		(* Execute FB *)
		fbCallMethod.nNumberOfInputArguments := nNoOfInputArgs;
		fbCallMethod.pInputArgInfo := ADR(aInputArgInfo);
		fbCallMethod.cbInputArgInfo := (SIZEOF(aInputArgInfo[1])*nNoOfInputArgs);
		fbCallMethod.pInputArgData := ADR(aInputData);
		fbCallMethod.cbInputArgData := nOffset;
		fbCallMethod.nNumberOfOutputArguments := nNoOfOutputArgs; 
		fbCallMethod.pOutputArgInfo := ADR(aOutputArgInfo); 
		fbCallMethod.cbOutputArgInfo := (SIZEOF(aOutputArgInfo[1]) * nNoOfOutputArgs); 
		fbCallMethod.pOutputArgInfoAndData := ADR(stUpdateVehicleReservationDataData.stOutput);
		fbCallMethod.cbOutputArgInfoAndData := SIZEOF(stUpdateVehicleReservationDataData.stOutput);
		
		stUpdateVehicleReservationDataData.iStatus := 1;
		bCallMethod := TRUE;
		
	ELSIF (stUpdateVehicleReservationDataData.iStatus = 1) THEN
		// Method call Completed...
		IF (eStateMethod = E_TrackClientState.Connected) THEN
			// Method call OK
			IF (stUpdateVehicleReservationDataData.stOutput.eStatus = E_MMServerStatus.eMMServerStatus_Success) THEN
				// Method returned OK
				stUpdateVehicleReservationDataData.iStatus := 2;
				// Trig vehicle data reading because data has changed
				M_VehicleToReadAdd(nVehicleID);
				
			ELSE
				// Method returned with error
				stUpdateVehicleReservationDataData.iStatus := 3;
				stUpdateVehicleReservationDataData.stOutput.sMessage;

			END_IF

		ELSIF (eStateMethod = E_TrackClientState.Error) THEN
			// Method call failed
			stUpdateVehicleReservationDataData.iStatus := 3;

		END_IF
		
	END_IF
ELSE
	M_CallUpdateVehicleReservationData := -1;
	RETURN;

END_IF

M_CallUpdateVehicleReservationData := stUpdateVehicleReservationDataData.iStatus;
END_METHOD

METHOD M_CallUpdateVehicleReworkData : INT
VAR_INPUT
	nVehicleID			: UINT;										(* Magnemotion Vehicle ID *)
	sCarrierID			: STRING(30);								(* Carrier ID *)
	bNOK				: BOOL;										(* TRUE signals that rework is required *)
END_VAR
VAR
END_VAR
IF (stUpdateVehicleReworkDataData.iStatus = 2) OR (stUpdateVehicleReworkDataData.iStatus = 3) THEN
	stUpdateVehicleReworkDataData.iStatus := 0;
END_IF

IF (bConnectedMethod AND NOT bBusyMethod) THEN
	IF (stUpdateVehicleReworkDataData.iStatus = 0) THEN
	(* Setup method calling parameters *)
		(* Method identifier *)
		sObjectIDentifier := stUpdateVehicleReworkDataData.sObjectID;
		sMethodIdentifier := stUpdateVehicleReworkDataData.sMethodID;
	
		(* Method Inputs *)
		stUpdateVehicleReworkDataData.stInput.sCarrierID := sCarrierID;
		stUpdateVehicleReworkDataData.stInput.bNOK := bNOK;
		
		(* Fill input data area with method arguments *)
		MEMSET(ADR(aInputData), 0 ,SIZEOF(aInputData));
		nOffset := 0;
		nOffset := nOffset + MEMCPY(ADR(aInputData)+nOffset, ADR(stUpdateVehicleReworkDataData.stInput),	MIN(SIZEOF(stUpdateVehicleReworkDataData.stInput), (SIZEOF(aInputData)-nOffset)) );
		(* Number of input arguments *)
		nNoOfInputArgs := stUpdateVehicleReworkDataData.iNoOfInputArgs;
		(* Set up input argument information *)
		MEMSET(ADR(aInputArgInfo), 0, SIZEOF(aInputArgInfo));
		aInputArgInfo[1].DataType := eUAType_String;
		aInputArgInfo[1].ValueRank := -1;	// -1: Scalar 
		aInputArgInfo[1].nLenData := SIZEOF(stUpdateVehicleReworkDataData.stInput.sCarrierID);
		aInputArgInfo[2].DataType := eUAType_Boolean;
		aInputArgInfo[2].ValueRank := -1;	// -1: Scalar 
		aInputArgInfo[2].nLenData := SIZEOF(stUpdateVehicleReworkDataData.stInput.bNOK);
		
		(* Method outputs *)
		(* Clear output data area *)
		(* Number of output arguments *)
		nNoOfOutputArgs := stUpdateVehicleReworkDataData.iNoOfOutputArgs;
		(* Set up output argument information *)
		MEMSET(ADR(aOutputArgInfo), 0, SIZEOF(aOutputArgInfo));
		aOutputArgInfo[1].DataType := eUAType_Uint16;
		aOutputArgInfo[1].ValueRank := -1;
		aOutputArgInfo[1].nLenData := SIZEOF(stUpdateVehicleReworkDataData.stOutput.eStatus);
		aOutputArgInfo[2].DataType := eUAType_String;
		aOutputArgInfo[2].ValueRank := -1;
		aOutputArgInfo[2].nLenData := SIZEOF(stUpdateVehicleReworkDataData.stOutput.sMessage);
		(* Set up output  *)
		MEMSET(ADR(stUpdateVehicleReworkDataData.stOutput), 0, SIZEOF(stUpdateVehicleReworkDataData.stOutput));
		stUpdateVehicleReworkDataData.stOutput.nNumberOfOutputArguments := nNoOfOutputArgs;
		stUpdateVehicleReworkDataData.stOutput.stOutputArgInfo[1] := aOutputArgInfo[1];
		stUpdateVehicleReworkDataData.stOutput.stOutputArgInfo[2] := aOutputArgInfo[2];
	
		(* Execute FB *)
		fbCallMethod.nNumberOfInputArguments := nNoOfInputArgs;
		fbCallMethod.pInputArgInfo := ADR(aInputArgInfo);
		fbCallMethod.cbInputArgInfo := (SIZEOF(aInputArgInfo[1])*nNoOfInputArgs);
		fbCallMethod.pInputArgData := ADR(aInputData);
		fbCallMethod.cbInputArgData := nOffset;
		fbCallMethod.nNumberOfOutputArguments := nNoOfOutputArgs; 
		fbCallMethod.pOutputArgInfo := ADR(aOutputArgInfo); 
		fbCallMethod.cbOutputArgInfo := (SIZEOF(aOutputArgInfo[1]) * nNoOfOutputArgs); 
		fbCallMethod.pOutputArgInfoAndData := ADR(stUpdateVehicleReworkDataData.stOutput);
		fbCallMethod.cbOutputArgInfoAndData := SIZEOF(stUpdateVehicleReworkDataData.stOutput);
		
		stUpdateVehicleReworkDataData.iStatus := 1;
		bCallMethod := TRUE;
		
	ELSIF (stUpdateVehicleReworkDataData.iStatus = 1) THEN
		// Method call Completed...
		IF (eStateMethod = E_TrackClientState.Connected) THEN
			// Method call OK
			IF (stUpdateVehicleReworkDataData.stOutput.eStatus = E_MMServerStatus.eMMServerStatus_Success) THEN
				// Method returned OK
				stUpdateVehicleReworkDataData.iStatus := 2;
				// Trig vehicle data reading because data has changed
				M_VehicleToReadAdd(nVehicleID);
								
			ELSE
				// Method returned with error
				stUpdateVehicleReworkDataData.iStatus := 3;
				stUpdateVehicleReworkDataData.stOutput.sMessage;
				
			END_IF
			
		ELSIF (eStateMethod = E_TrackClientState.Error) THEN
			// Method call failed
			stUpdateVehicleReworkDataData.iStatus := 3;

		END_IF
		
	END_IF
ELSE
	M_CallUpdateVehicleReworkData := -1;
	RETURN;

END_IF

M_CallUpdateVehicleReworkData := stUpdateVehicleReworkDataData.iStatus;
END_METHOD

METHOD PROTECTED M_CarrierIDToVehicleID : UINT
VAR_INPUT
	sCarrierID		: STRING(30);
END_VAR

VAR
	i: INT;
END_VAR

// Find vehicle with specified Carrier ID
FOR i := 1 TO MM_MAX_NUMBER_OF_VEHICLE_ELEMENTS BY 1 DO
	IF (aReadVehicleData[i].stVehicle.bDataValid) THEN
		IF (F_StringCompNoCase(aReadVehicleData[i].stVehicle.sCarrierID, sCarrierID) ) THEN
			M_CarrierIDToVehicleID := aReadVehicleData[i].stVehicle.nVehicleID;
			RETURN;
		END_IF
	END_IF
END_FOR

// Not found!
M_CarrierIDToVehicleID := 0;
END_METHOD

/// Check if a specified station index belongs to this cell
METHOD PROTECTED M_CheckStationIndex : BOOL
VAR_INPUT
	iStationNo		: UINT;
END_VAR
VAR
	i				: UINT;
END_VAR

FOR i := 1 TO 5 BY 1 DO
	IF (aStations[i].bPresent) THEN
		IF (iThisStationIndex[i] = iStationNo) THEN
			// Station index found
			M_CheckStationIndex := TRUE;
			RETURN;			
		END_IF
	END_IF
END_FOR

// Not found
M_CheckStationIndex := FALSE;
RETURN;
END_METHOD

/// Check if indexes are found for all specified stations
METHOD PROTECTED M_CheckStationsRead : BOOL
VAR
	i				: UINT;
	bReturn			: BOOL;
END_VAR

bReturn := TRUE;

FOR i := 1 TO 5 BY 1 DO
	IF (aStations[i].bPresent) THEN
		IF (iThisStationIndex[i] > 0) THEN
			// Station index found
		ELSE
			// Index for this station is not found!
			bReturn := FALSE;
			EXIT;
		END_IF
	END_IF
END_FOR

// Not found
M_CheckStationsRead := bReturn;
RETURN;
END_METHOD

/// Check if specified vehicle is Owned by this cell and is to be read (evet-driven reading)
METHOD PROTECTED M_CheckVehicleEventRead : BOOL
VAR_INPUT
	iVehicleNo		: UINT;		// MagneMotion Vehicle number
END_VAR
VAR
	i				: UINT;
	bVehicleOwned	: BOOL;
	bVehicleDoRead	: BOOL;
END_VAR

FOR i := 1 TO MM_MAX_NUMBER_OF_VEHICLE_ELEMENTS BY 1 DO
	IF (anVehiclesToRead[i] = iVehicleNo) THEN
		// Vehicle is found in to-read list
		M_CheckVehicleEventRead := TRUE;
		RETURN;
	END_IF

END_FOR

// Not found
M_CheckVehicleEventRead := FALSE;
RETURN;
END_METHOD

/// Check if specified vehicle is Owned by this cell
METHOD PROTECTED M_CheckVehicleOwned : BOOL
VAR_INPUT
	iVehicleNo		: UINT;		// MagneMotion Vehicle number
END_VAR
VAR
	i				: UINT;
END_VAR

FOR i := 1 TO MM_MAX_NUMBER_OF_VEHICLE_ELEMENTS BY 1 DO
	IF (aReadCellData.stCell.anVehicles[i] = iVehicleNo) THEN
		// Vehicle is found
		M_CheckVehicleOwned := TRUE;
		RETURN;
	END_IF
END_FOR

// Not found
M_CheckVehicleOwned := FALSE;
RETURN;
END_METHOD

/// Check if specified vehicle is survailed by this cell
METHOD PROTECTED M_CheckVehicleSurvail : BOOL
VAR_INPUT
	iVehicleNo		: UINT;		// MagneMotion Vehicle number
END_VAR
VAR
	i				: UINT;
END_VAR

FOR i := 1 TO MM_MAX_NUMBER_OF_VEHICLE_ELEMENTS BY 1 DO
	IF (anExtraVehicles[i] = iVehicleNo) THEN
		// Vehicle is found
		M_CheckVehicleSurvail := TRUE;
		RETURN;
	END_IF
END_FOR

// Not found
M_CheckVehicleSurvail := FALSE;
RETURN;
END_METHOD

METHOD M_ClearAll : BOOL
VAR_INPUT
END_VAR
VAR
	i	: UINT;
END_VAR

//Clear data on station(s)
FOR i:=1 TO 5 DO
	IF aStations[i].bPresent THEN
		// Station data
		aStations[i].stStationData1.nTicket := 0;
		aStations[i].stStationData1.nTicketSize := 0;
		aStations[i].stStationData1.CurrentPriority := 0;
		aStations[i].stStationData1.nCurrentVehicleID := 0;
		aStations[i].stStationData1.nReservedVehicleID := 0;
		aStations[i].stStationData2.nTicket := 0;
		aStations[i].stStationData2.nTicketSize := 0;
		aStations[i].stStationData2.CurrentPriority := 0;
		aStations[i].stStationData2.nCurrentVehicleID := 0;
		aStations[i].stStationData2.nReservedVehicleID := 0;
		
		// Station in/output
		bReadyStationIn[i] := FALSE;
		bReadyStationOut[i] := FALSE;

	END_IF
END_FOR

M_ClearAll := TRUE;
END_METHOD

METHOD PROTECTED M_CommandData
VAR_INPUT
END_VAR
VAR
	i			: USINT;
	iRes		: UINT;
END_VAR
// Handle the command data from OPC UA (stCommand)

CASE eCommandDataState OF
	// Init state
	E_CommandDataState.Undefined:
		eCommandDataState := E_CommandDataState.CheckRequest;		

	// Check command data request
	E_CommandDataState.CheckRequest:
		IF ((stCommand.ChangeRequest <> stStatus.ChangeStatus) AND (stCommand.ChangeRequest > 0)) THEN
			// Check if changes is allowed on mapping data (from LC)
			IF (stAdditionalDataIn.MESHandShakes.DataChangeStatusTransportStatus = stStatus.DataChange) THEN
// NOTE: Changed to match new LC software!!! - Hack!				
//				stStatus.ChangeAcknowledge := stCommand.ChangeRequest;
//				stStatus.DataChange := stStatus.DataChange + 1;
			
				// Find vehicle ID for specified Carrier ID
				iCommandDataVehicleID := M_CarrierIDToVehicleID(stCommand.CarrierID);
				IF ((iCommandDataVehicleID > 0) AND (iCommandDataVehicleID <= MM_MAX_NUMBER_OF_VEHICLE_ELEMENTS)) THEN
					// Specified vehicle found
					IF (F_StringCompNoCase(aReadVehicleData[iCommandDataVehicleID].stVehicle.sOwnerCell, sCellID)) THEN
						// Vehicle belongs to this cell
						stStatus.ValidRequest := TRUE;
						IF (stCommand.Ticket <= 0) THEN
							// Clear reservation data for this carrier (do not add reservation)
							eCommandDataState := E_CommandDataState.UpdateJobData;
						ELSE
							// Add reservation to track server
							eCommandDataState := E_CommandDataState.AddReservation;
						END_IF
					ELSE
						eCommandDataState := E_CommandDataState.Error;
					END_IF
				ELSE
					eCommandDataState := E_CommandDataState.Error;
				END_IF
			END_IF
		END_IF
		
	E_CommandDataState.AddReservation:
		iRes := M_CallAddReservation(	sStationID := stCommand.TargetStation,
										sCarrierID := stCommand.CarrierID,
										nTicket := stCommand.Ticket,
										nTicketSize := stCommand.CarriersInPackage,
										nPriority := stCommand.Priority 	);
		IF (iRes = 2) THEN
			// Success
			eCommandDataState := E_CommandDataState.UpdateJobData;
		ELSIF (iRes = 3) THEN
			// Error!
			F_LogLine('ERROR: AddReservation (Ticket: %d)', stCommand.Ticket);
			eCommandDataState := E_CommandDataState.Error;
		END_IF
	
	E_CommandDataState.UpdateJobData:
		iRes := M_CallUpdateVehicleReservationData(	nVehicleID := iCommandDataVehicleID,
													sTargetStationID := stCommand.TargetStation,
													sCarrierID := stCommand.CarrierID,
													nTicket := stCommand.Ticket,
													nCarriersInPackage := stCommand.CarriersInPackage,
													nPriority := stCommand.Priority,
													sJobID := stCommand.JobID 	);
		IF (iRes = 2) THEN
			// Success
			eCommandDataState := E_CommandDataState.Done;
		ELSIF (iRes = 3) THEN
			// Error!
			F_LogLine('ERROR: UpdateJobData (Ticket: %d)', stCommand.Ticket);
			eCommandDataState := E_CommandDataState.Error;
		END_IF
	
	E_CommandDataState.Done:
		stStatus.LatestTicket := stCommand.Ticket;
		stStatus.NumberOfCarriers := stCommand.CarriersInPackage;
		stStatus.ChangeStatus := stCommand.ChangeRequest;
// NOTE: Changed to match new LC software!!! - Hack!				
		stStatus.ChangeAcknowledge := stCommand.ChangeRequest;
		stStatus.DataChange := stStatus.DataChange + 1;
		eCommandDataState := E_CommandDataState.Undefined;
		
	E_CommandDataState.Error:
		stStatus.ValidRequest := FALSE;
		stStatus.ChangeStatus := stCommand.ChangeRequest;
// NOTE: Changed to match new LC software!!! - Hack!				
		stStatus.ChangeAcknowledge := stCommand.ChangeRequest;
		stStatus.DataChange := stStatus.DataChange + 1;
		eCommandDataState := E_CommandDataState.Undefined;
		
END_CASE
END_METHOD

/// Copy vehicle and ticket information from Source to Target and DELETES information on Source!!
METHOD PROTECTED M_CopyAndClearBufferData : BOOL
VAR_IN_OUT
	stSource		: ST_MMBuffer;
	stTarget		: ST_MMBuffer;
END_VAR

	// Update data for target location
	stTarget.nTicket := stSource.nTicket;
	stTarget.nTicketSize := stSource.nTicketSize;
	stTarget.CurrentPriority := stSource.CurrentPriority;
	stTarget.nReservedVehicleID := stSource.nReservedVehicleID;
	stTarget.nCurrentVehicleID := stSource.nCurrentVehicleID;
	// Clear data for source location
	stSource.nTicket := 0;
	stSource.nTicketSize := 0;
	stSource.CurrentPriority := 0;
	stSource.nCurrentVehicleID := 0;
	stSource.nReservedVehicleID := 0;
END_METHOD

/// Copy vehicle and ticket information from Source to Target and DELETES information on Source!!
METHOD PROTECTED M_CopyBufferData : BOOL
VAR_IN_OUT
	stSource		: ST_MMBuffer;
	stTarget		: ST_MMBuffer;
END_VAR

	// Update data for target location
	stTarget.nTicket := stSource.nTicket;
	stTarget.nTicketSize := stSource.nTicketSize;
	stTarget.CurrentPriority := stSource.CurrentPriority;
	stTarget.nReservedVehicleID := stSource.nReservedVehicleID;
	stTarget.nCurrentVehicleID := stSource.nCurrentVehicleID;
END_METHOD

// Set path to control from this cell
METHOD PUBLIC M_DefinePath : BOOL
VAR_INPUT
	nPathNo				: UINT;		// Path number
END_VAR
VAR
	i					: UINT;
	bFound				: BOOL;
END_VAR

bFound := FALSE;

IF ( (nPathNo > 0) AND (nPathNo <= MM_MAX_NUMBER_OF_PATH_ELEMENTS) ) THEN
	FOR i := 1 TO MM_MAX_NUMBER_OF_PATH_ELEMENTS BY 1 DO
		IF (aPaths[i] = nPathNo) THEN
			// Same path found
			IF (bFound) THEN
				// Already added to list, but found again, delete old value
				aPaths[i] := 0;
			END_IF
			bFound := TRUE;
		ELSIF ( (aPaths[i] = 0) AND NOT bFound ) THEN
			// Free spot found, assign value
			aPaths[i] := nPathNo;
			bFound := TRUE;
		END_IF
	END_FOR
END_IF

M_DefinePath := bFound;
END_METHOD

METHOD PUBLIC M_DefinePathSegment : BOOL
VAR_INPUT
	nPathSegmentNo	: UINT;
	nPathID			: UINT;		// Path number
	rPositionBegin	: REAL;		// Distance on the specified path to begin segment
	rPositionEnd	: REAL;		// Distance on the specified path to end segment
END_VAR
// Check if data is valid
IF ( (nPathID > 0) AND (rPositionBegin >= 0.0) AND (rPositionEnd > rPositionBegin) ) THEN
	IF (nPathSegmentNo = 1) THEN
		stExitPointSeg1LocBegin.nPathID := nPathID;
		stExitPointSeg1LocBegin.fPosition := rPositionBegin;
		stExitPointSeg1LocEnd.nPathID := nPathID;
		stExitPointSeg1LocEnd.fPosition := rPositionEnd;
		M_DefinePathSegment := TRUE;
		
	ELSIF (nPathSegmentNo = 2) THEN
		stExitPointSeg2LocBegin.nPathID := nPathID;
		stExitPointSeg2LocBegin.fPosition := rPositionBegin;
		stExitPointSeg2LocEnd.nPathID := nPathID;
		stExitPointSeg2LocEnd.fPosition := rPositionEnd;
		M_DefinePathSegment := TRUE;
		
	ELSE
		M_DefinePathSegment := FALSE;
		
	END_IF

ELSE
	M_DefinePathSegment := FALSE;
	
END_IF
END_METHOD

// Set data for traffic light
METHOD PUBLIC M_DefineStation : BOOL
VAR_INPUT
	nStationNo			: UINT(1..5);
	sStationID			: STRING(30);
	nLoc1PathID			: UINT;		// Path number for input location
	rLoc1Position		: REAL;		// Distance on the specified path for input location
	nLoc2PathID			: UINT;		// Path number for output location (0 if single station)
	rLoc2Position		: REAL;		// Distance on the specified path for output location (0.0 if single station)
	nLocDecPathID		: UINT;		// Path number for decision point location
	rLocDecPosition		: REAL;		// Distance on the specified path for decision point location
	nPreBufferSize		: UINT;		// Size of pre buffer (number of positions)
	nPostBufferSize		: UINT;		// Size of post buffer (number of positions)
END_VAR
VAR
	i					: UINT;
	bReInit				: BOOL;
END_VAR
IF ( (nLoc1PathID > 0) AND (rLoc1Position >= 0.0) AND
//	 (nLoc2PathID > 0) AND (rLoc2Position >= 0.0) AND	// Allow single position stations!
	 (nLocDecPathID > 0) AND (rLocDecPosition >= 0.0) AND 
	 (nStationNo >= 1) AND (nStationNo <= 5) AND
	 (sStationID <> '') ) THEN
	
	IF ( (aStations[nStationNo].sStationID <> sStationID) OR
		 (aStations[nStationNo].stStationData1.stLocation.nPathID <> nLoc1PathID) OR
		 (aStations[nStationNo].stStationData1.stLocation.fPosition <> rLoc1Position) OR
		 (aStations[nStationNo].stStationData2.stLocation.nPathID <> nLoc2PathID) OR
		 (aStations[nStationNo].stStationData2.stLocation.fPosition <> rLoc2Position) OR
		 (aStations[nStationNo].stDecisionLocation.nPathID <> nLocDecPathID) OR
		 (aStations[nStationNo].stDecisionLocation.fPosition <> rLocDecPosition) OR
		 (aStations[nStationNo].bPresent = FALSE) ) THEN
		
		bReInit := TRUE;
	END_IF

	aStations[nStationNo].sStationID := sStationID;
	aStations[nStationNo].stStationData1.stLocation.nPathID := nLoc1PathID;
	aStations[nStationNo].stStationData1.stLocation.fPosition := rLoc1Position;
	IF (nLoc1PathID > 0) THEN
		aStations[nStationNo].stStationData1.bPresent := TRUE;
	ELSE
		aStations[nStationNo].stStationData1.bPresent := FALSE;		
	END_IF
	aStations[nStationNo].stStationData2.stLocation.nPathID := nLoc2PathID;
	aStations[nStationNo].stStationData2.stLocation.fPosition := rLoc2Position;
	IF (nLoc2PathID > 0) THEN
		aStations[nStationNo].stStationData2.bPresent := TRUE;
	ELSE
		aStations[nStationNo].stStationData2.bPresent := FALSE;		
	END_IF
	aStations[nStationNo].stDecisionLocation.nPathID := nLocDecPathID;
	aStations[nStationNo].stDecisionLocation.fPosition := rLocDecPosition;

	// Buffers	
	FOR i := 1 TO MM_MAX_BUFFER_INDEX BY 1 DO
		IF ( (aStations[nStationNo].astPreBuffer[i].bPresent <> (i <= nPreBufferSize)) OR
			 (aStations[nStationNo].astPostBuffer[i].bPresent <> (i <= nPostBufferSize)) ) THEN
			bReInit := TRUE;
		END_IF
		aStations[nStationNo].astPreBuffer[i].bPresent := (i <= nPreBufferSize);
		aStations[nStationNo].astPostBuffer[i].bPresent := (i <= nPostBufferSize);
	END_FOR
	aStations[nStationNo].bPresent := TRUE;
	
	M_DefineStation := TRUE;
ELSE
	M_DefineStation := FALSE;
END_IF
END_METHOD

// Set data for traffic light
METHOD PUBLIC M_DefineStationBufferAdjust : BOOL
VAR_INPUT
	nStationNo			: UINT(1..5);
	rPreBufferAdjust	: REAL;		// Distance to adjust pre-buffer position (M) - Should be negative for pre-buffer
	rPostBufferAdjust	: REAL;		// Distance to adjust post-buffer position (M) - Should be negative for pre-buffer
END_VAR
VAR
END_VAR
IF ( (nStationNo > 0) AND (nStationNo <= 5) ) THEN
	IF (aStations[nStationNo].bPresent) THEN
		// Station defined
		aStationPreBufAdj[nStationNo] := rPreBufferAdjust;
		aStationPostBufAdj[nStationNo] := rPostBufferAdjust;
		M_DefineStationBufferAdjust := TRUE;
	ELSE
		// Station not defined
		M_DefineStationBufferAdjust := FALSE;
	END_IF
ELSE
	// Outside range
	M_DefineStationBufferAdjust := FALSE;
END_IF
END_METHOD

// Set data for traffic light
METHOD PUBLIC M_DefineTrafficLight : BOOL
VAR_INPUT
	nTrafficLightNo	: UINT;
	nPathID			: UINT;		// Path number
	rPosition		: REAL;		// Distance on the specified path
END_VAR

IF ((nTrafficLightNo > 0) AND (nPathID > 0) AND (rPosition >= 0.0)) THEN
	IF (nTrafficLightNo = 1) THEN
		stTrafficLightLocation.nPathID := nPathID;
		stTrafficLightLocation.fPosition := rPosition;
		M_DefineTrafficLight := TRUE;

	ELSIF (nTrafficLightNo = 2) THEN
		stTrafficLight2Location.nPathID := nPathID;
		stTrafficLight2Location.fPosition := rPosition;
		M_DefineTrafficLight := TRUE;

	ELSE
		M_DefineTrafficLight := FALSE;
		
	END_IF
ELSE
	M_DefineTrafficLight := FALSE;
	
END_IF
END_METHOD

// Set data for enable/disable station
METHOD PUBLIC M_EnableStation : BOOL
VAR_INPUT
	nStationNo			: UINT(1..5);
	bPresent			: BOOL;
END_VAR
VAR
	i					: UINT;
END_VAR
IF (nStationNo <= 5) THEN
	aStations[nStationNo].bPresent := bPresent;
	
	M_EnableStation := TRUE;
ELSE
	M_EnableStation := FALSE;
END_IF
END_METHOD

METHOD PROTECTED M_ErrorWarning
VAR_INPUT
END_VAR
VAR
	bDataChange:BOOL;
END_VAR

bDataChange S= 
M_ErrorWarningObj(arErrorWaringData:= stErrorWarning.ErrorWarningData,
	bActive:= eTrackState = E_TrackState.Error, 
	iErrorWarningType:= 2, 
	diErrorWarningID:= E_AlarmCategory.TrackClient + 0, 
	sDeviceID:= 'Track Client',
	iSeverity:= 2, 
	iNativeID:= 0, 
	sNativeMessage:= 'Error State Machine');
	
bDataChange S= 
M_ErrorWarningObj(arErrorWaringData:= stErrorWarning.ErrorWarningData,
	bActive:= eStateMethod = E_TrackState.Error, 
	iErrorWarningType:= 2, 
	diErrorWarningID:= E_AlarmCategory.TrackClient + 1, 
	sDeviceID:= 'Track Client',
	iSeverity:= 2, 
	iNativeID:= 0, 
	sNativeMessage:= 'Error State Machine Method');
	
bDataChange S= 
M_ErrorWarningObj(arErrorWaringData:= stErrorWarning.ErrorWarningData,
	bActive:= eStateNode = E_TrackState.Error, 
	iErrorWarningType:= 2, 
	diErrorWarningID:= E_AlarmCategory.TrackClient + 2, 
	sDeviceID:= 'Track Client',
	iSeverity:= 2, 
	iNativeID:= 0, 
	sNativeMessage:= 'Error State Machine Node ADS');


stErrorWarning.DataChange := stErrorWarning.DataChange + TO_UINT(bDataChange);
bDataChange := FALSE;
END_METHOD

METHOD M_ErrorWarningObj : BOOL
VAR_INPUT
	bActive				: BOOL;
	iErrorWarningType	: UINT;
	diErrorWarningID 	: UDINT;
	sDeviceID			: STRING(30);
	iSeverity			: UINT;
	iNativeID			: UDINT;
	sNativeMessage		: STRING(80);
END_VAR
VAR_IN_OUT
	arErrorWaringData	: ARRAY [1..255] OF ST_ErrorWarningDataX;
END_VAR
VAR
	iFoundPos			: UINT;
	i					: UINT;
	j					: UINT;
END_VAR
//Look through array to find existing record(s)
FOR i := 1 TO 255 DO
	IF arErrorWaringData[i].ErrorWarningID = 0 THEN
		EXIT;
	END_IF
	//Existing alarm - first
	IF arErrorWaringData[i].ErrorWarningID = diErrorWarningID AND iFoundPos = 0 THEN
		iFoundPos := i;
	//Multiple records - delete
	ELSIF arErrorWaringData[i].ErrorWarningID = diErrorWarningID AND iFoundPos <> 0 THEN
		MEMSET(ADR(arErrorWaringData[i]), 0, SIZEOF(arErrorWaringData[i]));
		M_ErrorWarningObj := TRUE;
	END_IF
END_FOR

//Alarm high
IF bActive THEN
	//New alarm
	IF iFoundPos = 0 THEN
		arErrorWaringData[i].ErrorWarningType := iErrorWarningType;
		arErrorWaringData[i].DeviceID := sDeviceID;
		arErrorWaringData[i].Severity := iSeverity;
		arErrorWaringData[i].NativeID := iNativeID;
		arErrorWaringData[i].NativeMessage := sNativeMessage;
		arErrorWaringData[i].ErrorWarningID := diErrorWarningID;
		arErrorWaringData[i].DateTime := SYSTEMTIME_TO_STRING(fbGetTime.TIMESTR);
		M_ErrorWarningObj := TRUE;
	END_IF
	
//Alarm low
ELSIF NOT bActive AND iFoundPos <> 0 THEN
	MEMSET(ADR(arErrorWaringData[iFoundPos]), 0, SIZEOF(arErrorWaringData[iFoundPos]));
	M_ErrorWarningObj := TRUE;
END_IF

//Defrag
IF M_ErrorWarningObj THEN
	FOR i:= 1 TO 254 DO
		//Find first empty spot
		IF arErrorWaringData[i].ErrorWarningID = 0 THEN
			//Find first record
			FOR j:= i TO 255 DO
				IF arErrorWaringData[j].ErrorWarningID <> 0 THEN
					//Move to empty spot
					arErrorWaringData[i] := arErrorWaringData[j];
					MEMSET(ADR(arErrorWaringData[j]), 0, SIZEOF(arErrorWaringData[j]));
					EXIT;
				END_IF
			END_FOR
		END_IF
		//No more records
		IF j >= 255 THEN
			RETURN;
		END_IF
	END_FOR
END_IF
END_METHOD

/// Add vehicle to be survailed
METHOD PROTECTED M_ExtraVehicleAdd : BOOL
VAR_INPUT
	iVehicleNo		: UINT;
END_VAR
VAR
	i				: UINT;
	bAdded			: BOOL;
	bRemoved		: BOOL;
END_VAR

FOR i := 1 TO MM_MAX_NUMBER_OF_VEHICLE_ELEMENTS BY 1 DO
	// Check if already excists in list
	IF (anExtraVehicles[i] = iVehicleNo) THEN
		anExtraVehicles[i] := 0;
		bRemoved := TRUE;
	END_IF
	// Add to list
	IF ( (NOT bAdded) AND (anExtraVehicles[i] = 0) ) THEN
		anExtraVehicles[i] := iVehicleNo;
		bAdded := TRUE;
	END_IF
	// Check if finished
	IF (bAdded AND bRemoved) THEN
		M_ExtraVehicleAdd := TRUE;
		RETURN;
	END_IF
	
END_FOR

IF (bAdded) THEN
	// Added
	M_ExtraVehicleAdd := TRUE;
	RETURN;
ELSE
	// NOT Added (list is maybe full!)
	M_ExtraVehicleAdd := FALSE;
	RETURN;	
END_IF
END_METHOD

/// Remove vehicle from surveillance list
METHOD PROTECTED M_ExtraVehicleRemove : BOOL
VAR_INPUT
	iVehicleNo		: UINT;
END_VAR
VAR
	i				: UINT;
END_VAR

FOR i := 1 TO MM_MAX_NUMBER_OF_VEHICLE_ELEMENTS BY 1 DO
	IF (anExtraVehicles[i] = iVehicleNo) THEN
		anExtraVehicles[i] := 0;
		M_ExtraVehicleRemove := TRUE;
		RETURN;
	END_IF
END_FOR

// Not found
M_ExtraVehicleRemove := FALSE;
RETURN;
END_METHOD

METHOD PROTECTED M_Init : BOOL
VAR_INPUT
END_VAR
VAR
	i : UINT;
	sTemp : STRING;
END_VAR
IF (NOT bInitDone) THEN
// Client information to stations
	FOR i := 1 TO 5 BY 1 DO
		aStations[i].sCellID := sCellID;
	END_FOR

// OPC UA Method calling information
	(* Use no encryption *)
	stConnectInfoMethod.eSecurityMode 			:= eUASecurityMsgMode_None;
	(*  *)
	stConnectInfoMethod.eSecurityPolicyUri		:= eUASecurityPolicy_None;
	(* USe TCP transport profile *)
	stConnectInfoMethod.eTransportProfileUri	:= eUATransportProfileUri_UATcp;
	(* Application name *)
	stConnectInfoMethod.sApplicationName		:= '';
	(* Connection timeout *)
	stConnectInfoMethod.tConnectTimeout			:= T#1M;
	(* Session timeout *)
	stConnectInfoMethod.tSessionTimeout			:= T#10M;
	(* Method node ID *)
	stObjectNodeID.eIdentifierType				:= E_UAIdentifierType.eUAIdentifierType_String;
	stMethodNodeID.eIdentifierType				:= E_UAIdentifierType.eUAIdentifierType_String;
	(* Method data *)
	M_InitMethodData();
	
// OPC UA Node reading information
	(* Use no encryption *)
	stConnectInfoNodes.eSecurityMode 			:= eUASecurityMsgMode_None;
	(*  *)
	stConnectInfoNodes.eSecurityPolicyUri		:= eUASecurityPolicy_None;
	(* USe TCP transport profile *)
	stConnectInfoNodes.eTransportProfileUri		:= eUATransportProfileUri_UATcp;
	(* Application name *)
	stConnectInfoNodes.sApplicationName			:= '';
	(* Connection timeout *)
	stConnectInfoNodes.tConnectTimeout			:= T#1M;
	(* Session timeout *)
	stConnectInfoNodes.tSessionTimeout			:= T#10M;

	
	bInitDone := TRUE;
END_IF
END_METHOD

METHOD PROTECTED M_InitMethodData : BOOL

(* Method data *)
stAddStationDoubleData.iStatus				:= 0;
stAddStationSingleData.iStatus				:= 0;
stEnableStationData.iStatus					:= 0;
stRemoveStationData.iStatus					:= 0;

stGetCellIndexData.iStatus					:= 0;

stAddPathData.iStatus						:= 0;
stRemovePathData.iStatus					:= 0;
stStartPathData.iStatus						:= 0;
stResetPathData.iStatus						:= 0;
stSuspendPathData.iStatus					:= 0;
stResumePathData.iStatus					:= 0;

stAddTrafficLightData.iStatus				:= 0;
stRemoveTrafficLightData.iStatus			:= 0;
stTrafficLightColorData.iStatus				:= 0;
stSetTrafficLightColorData.iStatus			:= 0;

stMoveToStationInData.iStatus				:= 0;
stMoveToStationOutData.iStatus				:= 0;
stMoveToPositionData.iStatus				:= 0;
stMoveToBufferData.iStatus					:= 0;
stMoveToDecisionPointData.iStatus			:= 0;
stMoveToScannerData.iStatus					:= 0;

//stUpdateVehicleDataData.iStatus			:= 0;
stUpdateVehicleReservationDataData.iStatus	:= 0;
stUpdateVehicleMappingDataData.iStatus		:= 0;
stUpdateVehicleReworkDataData.iStatus		:= 0;
END_METHOD

METHOD PROTECTED M_InitNodeData : BOOL
VAR
	i				: UINT;
	sPrefix 		: STRING;
	
	bReturn			: BOOL;
END_VAR

(* Node data, init to use string identifier and set namespace index *)
FOR i:=1 TO nMaxNodeIDsInList BY 1 DO
	aNodeIDs[i].eIdentifierType := eUAIdentifierType_String;
	aNodeIDs[i].nNamespaceIndex := nNameSpaceIndexNodes;
END_FOR

nNoOfNodes := 0;
cbDataTotal := 0;

// TEST
//eReadType := E_OPC_NodeType.Nodes;
//iReadIndex := 1;

// Comm type selection
CASE eReadType OF
	E_OPC_NodeType.Vehicles:
		// Select vehicle to read data from
		REPEAT
			iReadIndex := iReadIndex+1;
			IF (iReadIndex > MM_MAX_NUMBER_OF_VEHICLE_ELEMENTS) THEN
				EXIT;
			END_IF
			UNTIL (aReadCellData.stCell.anVehicles[iReadIndex] > 0)
		END_REPEAT
		IF (iReadIndex <= MM_MAX_NUMBER_OF_VEHICLE_ELEMENTS) THEN
			// Build remote symbol name
			sPrefix := CONCAT(sObjectIDentifier, '.stTrackStatus');
			// Data pointer for received data
			pReadNodeData := ADR(aReadVehicleData[iReadIndex]);
			// Header data size
			cbDataTotal := SIZEOF(aReadVehicleData[iReadIndex].stReadListReturnInfo);
			
			// Specify nodes to read by variable name
			nNoOfNodes := nNoOfNodes + 1;
			aNodeIDs[nNoOfNodes].sIdentifier := CONCAT(sPrefix, '.aVehicles[');
			aNodeIDs[nNoOfNodes].sIdentifier := CONCAT(aNodeIDs[nNoOfNodes].sIdentifier, UINT_TO_STRING(aReadCellData.stCell.anVehicles[iReadIndex]));
			aNodeIDs[nNoOfNodes].sIdentifier := CONCAT(aNodeIDs[nNoOfNodes].sIdentifier, ']');
			acbDatas[nNoOfNodes] := SIZEOF(aReadVehicleData[iReadIndex]);
			cbDataTotal := cbDataTotal + acbDatas[nNoOfNodes];
			bReturn := TRUE;
		ELSE
			// Read next type
			iReadIndex := 0;
			eReadType := E_OPC_NodeType.Paths;
			bReturn := FALSE;
		END_IF			
		
	E_OPC_NodeType.Paths:
		// Select path to read data from
		REPEAT
			iReadIndex := iReadIndex+1;
			IF (iReadIndex > MM_MAX_NUMBER_OF_PATH_ELEMENTS) THEN
				EXIT;
			END_IF
			UNTIL (abControlledPaths[i])
		END_REPEAT
		IF (iReadIndex <= MM_MAX_NUMBER_OF_PATH_ELEMENTS) THEN
			// Build remote symbol name
			sPrefix := CONCAT(sObjectIDentifier, '.stTrackStatus');
			// Data pointer for received data
			pReadNodeData := ADR(aReadPathData[iReadIndex]);
			// Header data size
			cbDataTotal := SIZEOF(aReadPathData[iReadIndex].stReadListReturnInfo);
			
			// Specify nodes to read by variable name
			nNoOfNodes := nNoOfNodes + 1;
			aNodeIDs[nNoOfNodes].sIdentifier := CONCAT(sPrefix, '.aPaths[');
			aNodeIDs[nNoOfNodes].sIdentifier := CONCAT(aNodeIDs[nNoOfNodes].sIdentifier, UINT_TO_STRING(iReadIndex));
			aNodeIDs[nNoOfNodes].sIdentifier := CONCAT(aNodeIDs[nNoOfNodes].sIdentifier, ']');
			acbDatas[nNoOfNodes] := SIZEOF(aReadPathData[iReadIndex]);
			cbDataTotal := cbDataTotal + acbDatas[nNoOfNodes];
			bReturn := TRUE;
		ELSE
			// Read next type
			iReadIndex := 0;
			eReadType := E_OPC_NodeType.Stations;
			bReturn := FALSE;
		END_IF
		
	E_OPC_NodeType.Stations:
		// Select Station to read data from
		iReadIndex := iReadIndex+1;
		IF (iReadIndex <= MM_MAX_NUMBER_OF_STATION_ELEMENTS) THEN
			// Build remote symbol name
			sPrefix := CONCAT(sObjectIDentifier, '.stTrackStatus');
			// Data pointer
			pReadNodeData := ADR(aReadStationData[iReadIndex]);
			
			// Header data
			cbDataTotal := SIZEOF(aReadStationData[iReadIndex].stReadListReturnInfo);
			
			// Specify nodes to read by variable name
			nNoOfNodes := nNoOfNodes + 1;
			aNodeIDs[nNoOfNodes].sIdentifier := CONCAT(sPrefix, '.aStations[');
			aNodeIDs[nNoOfNodes].sIdentifier := CONCAT(aNodeIDs[nNoOfNodes].sIdentifier, UINT_TO_STRING(iReadIndex));
			aNodeIDs[nNoOfNodes].sIdentifier := CONCAT(aNodeIDs[nNoOfNodes].sIdentifier, ']');
			acbDatas[nNoOfNodes] := SIZEOF(aReadStationData[iReadIndex].stStationData);
			cbDataTotal := cbDataTotal + acbDatas[nNoOfNodes];
			bReturn := TRUE;
		ELSE
			// Read next type
			iReadIndex := 0;
			eReadType := E_OPC_NodeType.Cells;
			bReturn := FALSE;
		END_IF
		
	E_OPC_NodeType.Cells:
		// Select cell status to read data from
		iReadIndex := iThisCellIndex;
		IF (iReadIndex > 0 AND iReadIndex <= MM_MAX_NUMBER_OF_STATION_ELEMENTS) THEN
			// Build remote symbol name
			sPrefix := CONCAT(sObjectIDentifier, '.stTrackStatus');
			// Data pointer
			pReadNodeData := ADR(aReadCellData);
			
			// Header data
			cbDataTotal := SIZEOF(aReadCellData.stReadListReturnInfo);
			
			// Specify nodes to read by variable name
			nNoOfNodes := nNoOfNodes + 1;
			aNodeIDs[nNoOfNodes].sIdentifier := CONCAT(sPrefix, '.aCells[');
			aNodeIDs[nNoOfNodes].sIdentifier := CONCAT(aNodeIDs[nNoOfNodes].sIdentifier, UINT_TO_STRING(iReadIndex));
			aNodeIDs[nNoOfNodes].sIdentifier := CONCAT(aNodeIDs[nNoOfNodes].sIdentifier, ']');
			acbDatas[nNoOfNodes] := SIZEOF(aReadCellData.stCell);
			cbDataTotal := cbDataTotal + acbDatas[nNoOfNodes]; 
			bReturn := TRUE;

			// continue to next type after this read!
			iReadIndex := 0;
			eReadType := E_OPC_NodeType.Vehicles;
		ELSE
			// Read next type
			iReadIndex := 0;
			eReadType := E_OPC_NodeType.Vehicles;
			bReturn := FALSE;
		END_IF
	
END_CASE
END_METHOD

METHOD PROTECTED M_InitNodeData_ADS : BOOL
VAR
	i				: UINT;
	sPrefix 		: STRING;
	
	bReturn			: BOOL;
END_VAR

nNoOfNodes := 0;
cbDataTotal := 0;

// TEST NEW
IF ( (nDecisionPointVehicleNo > 0) AND bReadDecPointVehicle ) THEN
	// Read data from vehicle at decision point (Higher priority!)
	// Build remote symbol name
	sPrefix := CONCAT(sObjectIDentifier, '.stTrackStatus');
	// Data pointer for received data
	pReadNodeData := ADR(aReadVehicleData[nDecisionPointVehicleNo].stVehicle);
	// Header data size
	cbDataTotal := SIZEOF(aReadVehicleData[nDecisionPointVehicleNo].stVehicle);
	
	// Specify nodes to read by variable name
	sTrackServerSymbol := CONCAT(sPrefix, '.aVehicles[');
	sTrackServerSymbol := CONCAT(sTrackServerSymbol, UINT_TO_STRING(nDecisionPointVehicleNo));
	sTrackServerSymbol := CONCAT(sTrackServerSymbol, ']');

	// Remove this vehicle from the event-driven reading list (to make sure it is not continously read!)
	M_VehicleToReadRemove(nDecisionPointVehicleNo);
				
	bReadDecPointVehicle := FALSE;	// Done in M_StateMachineNode_ADS
	bReadDecPointVehicleBusy := TRUE;
	bReturn := TRUE;

	M_InitNodeData_ADS := bReturn;
	RETURN;
END_IF
// END TEST NEW

// Comm type selection
CASE eReadType OF
	E_OPC_NodeType.Vehicles:
		IF ( (nDecisionPointVehicleNo > 0) AND bReadDecPointVehicle ) THEN
			// Read data from vehicle at decision point (Higher priority!)
			// Build remote symbol name
			sPrefix := CONCAT(sObjectIDentifier, '.stTrackStatus');
			// Data pointer for received data
			pReadNodeData := ADR(aReadVehicleData[nDecisionPointVehicleNo].stVehicle);
			// Header data size
			cbDataTotal := SIZEOF(aReadVehicleData[nDecisionPointVehicleNo].stVehicle);
			
			// Specify nodes to read by variable name
			sTrackServerSymbol := CONCAT(sPrefix, '.aVehicles[');
			sTrackServerSymbol := CONCAT(sTrackServerSymbol, UINT_TO_STRING(nDecisionPointVehicleNo));
			sTrackServerSymbol := CONCAT(sTrackServerSymbol, ']');

			// Remove this vehicle from the event-driven reading list (to make sure it is not continously read!)
			M_VehicleToReadRemove(nDecisionPointVehicleNo);
				
			bReadDecPointVehicle := FALSE;	// Done in M_StateMachineNode_ADS
			bReadDecPointVehicleBusy := TRUE;
			bReturn := TRUE;			
		ELSE
	// NEW!!!
			// NOTE: iReadIndex is MagneMotion vehicle No
			REPEAT
				iReadIndex := iReadIndex + 1;
				IF (M_CheckVehicleOwned(iReadIndex)) THEN
					// Vehicle is owned by this cell... Read data from Track Server for this vehicle
					IF (M_CheckVehicleEventRead(iReadIndex)) THEN
						// Vehicle data is selected to be read! (event-based reading)
						EXIT;
					END_IF
				ELSIF (M_CheckVehicleSurvail(iReadIndex)) THEN
					// Vehicle is survailed by this cell (read data continously!)... Read data from Track Server for this vehicle
					EXIT;
				ELSIF (iReadIndex <> nDecisionPointVehicleNo) THEN
					// Not owned or surveilled or being handled by decision point. Delete any previous read data
					IF (iReadIndex > 0 AND iReadIndex <= MM_MAX_NUMBER_OF_VEHICLE_ELEMENTS) THEN
						aReadVehicleData[iReadIndex].stVehicle.bDataValid := FALSE;
					END_IF
				END_IF
				UNTIL (iReadIndex >= MM_MAX_NUMBER_OF_VEHICLE_ELEMENTS)
			END_REPEAT
			
			IF (iReadIndex <= MM_MAX_NUMBER_OF_VEHICLE_ELEMENTS) THEN
				// Build remote symbol name
				sPrefix := CONCAT(sObjectIDentifier, '.stTrackStatus');
				// Data pointer for received data
				pReadNodeData := ADR(aReadVehicleData[iReadIndex].stVehicle);
				// Header data size
				cbDataTotal := SIZEOF(aReadVehicleData[iReadIndex].stVehicle);
				
				// Specify nodes to read by variable name
				sTrackServerSymbol := CONCAT(sPrefix, '.aVehicles[');
				sTrackServerSymbol := CONCAT(sTrackServerSymbol, UINT_TO_STRING(iReadIndex));
				sTrackServerSymbol := CONCAT(sTrackServerSymbol, ']');
				
				// Remove this vehicle from the event-driven reading list
				M_VehicleToReadRemove(iReadIndex);
				
				bReturn := TRUE;
			ELSE
				// Read next type
				iReadIndex := 0;
				eReadType := E_OPC_NodeType.Paths;
				bReturn := FALSE;
			END_IF
	// NEW END!!!	
			// Select vehicle to read data from (only the vehicles this cell is responsible for)
(*			REPEAT
				iReadIndex := iReadIndex+1;
				IF (iReadIndex > MM_MAX_NUMBER_OF_VEHICLE_ELEMENTS) THEN
					EXIT;
				END_IF
				UNTIL (aReadCellData.stCell.anVehicles[iReadIndex] > 0)
			END_REPEAT
			IF (iReadIndex <= MM_MAX_NUMBER_OF_VEHICLE_ELEMENTS) THEN
				// Build remote symbol name
				sPrefix := CONCAT(sObjectIDentifier, '.stTrackStatus');
				// Data pointer for received data
				pReadNodeData := ADR(aReadVehicleData[aReadCellData.stCell.anVehicles[iReadIndex]].stVehicle);
				// Header data size
				cbDataTotal := SIZEOF(aReadVehicleData[aReadCellData.stCell.anVehicles[iReadIndex]].stVehicle);
				
				// Specify nodes to read by variable name
				sTrackServerSymbol := CONCAT(sPrefix, '.aVehicles[');
				sTrackServerSymbol := CONCAT(sTrackServerSymbol, UINT_TO_STRING(aReadCellData.stCell.anVehicles[iReadIndex]));
				sTrackServerSymbol := CONCAT(sTrackServerSymbol, ']');
				bReturn := TRUE;
			ELSE
				// Read next type
				iReadIndex := 0;
				eReadType := E_OPC_NodeType.Paths;
				bReturn := FALSE;
			END_IF		*)
		END_IF
		
	E_OPC_NodeType.Paths:
		// Select path to read data from
		REPEAT
			iReadIndex := iReadIndex+1;
			IF (iReadIndex > MM_MAX_NUMBER_OF_PATH_ELEMENTS) THEN
				EXIT;
			END_IF
			UNTIL (abControlledPaths[iReadIndex])
		END_REPEAT
		IF ((iReadIndex <= MM_MAX_NUMBER_OF_PATH_ELEMENTS) AND NOT tonSkipPathRead.Q) THEN	// Skip path reading when paths are started!
			// Build remote symbol name
			sPrefix := CONCAT(sObjectIDentifier, '.stTrackStatus');
			// Data pointer for received data
			pReadNodeData := ADR(aReadPathData[iReadIndex].stPathData);
			// Header data size
			cbDataTotal := SIZEOF(aReadPathData[iReadIndex].stPathData);
			
			// Specify nodes to read by variable name
			sTrackServerSymbol := CONCAT(sPrefix, '.aPaths[');
			sTrackServerSymbol := CONCAT(sTrackServerSymbol, UINT_TO_STRING(iReadIndex));
			sTrackServerSymbol := CONCAT(sTrackServerSymbol, ']');
			bReturn := TRUE;
		ELSE
			// Read next type
			iReadIndex := 0;
			eReadType := E_OPC_NodeType.Stations;
			bReturn := FALSE;
		END_IF
		
	E_OPC_NodeType.Stations:
		// Select Station to read data from
// TEST
		IF (M_CheckStationsRead()) THEN
			// Index for station data from track server has been found... Only read these stations
			REPEAT
				iReadIndex := iReadIndex+1;
				IF (iReadIndex > MM_MAX_NUMBER_OF_STATION_ELEMENTS) THEN
					EXIT;
				END_IF
				UNTIL (M_CheckStationIndex(iReadIndex))
			END_REPEAT
		ELSE
			// Index for station data from track server has NOT been found... Read data from all stations
			iReadIndex := iReadIndex + 1;
		END_IF
// TEST END
//		iReadIndex := iReadIndex+1;
		IF (iReadIndex <= MM_MAX_NUMBER_OF_STATION_ELEMENTS) THEN
			// Build remote symbol name
			sPrefix := CONCAT(sObjectIDentifier, '.stTrackStatus');
			// Data pointer
			pReadNodeData := ADR(aReadStationData[iReadIndex].stStationData);
			// Header data
			cbDataTotal := SIZEOF(aReadStationData[iReadIndex].stStationData);
			
			// Specify nodes to read by variable name
			sTrackServerSymbol := CONCAT(sPrefix, '.aStations[');
			sTrackServerSymbol := CONCAT(sTrackServerSymbol, UINT_TO_STRING(iReadIndex));
			sTrackServerSymbol := CONCAT(sTrackServerSymbol, ']');
			bReturn := TRUE;
		ELSE
			// Read next type
			iReadIndex := 0;
			eReadType := E_OPC_NodeType.Cells;
			bReturn := FALSE;
		END_IF
	
	E_OPC_NodeType.Cells:
		// Select Station to read data from
		iReadIndex := iThisCellIndex;
		IF (iReadIndex > 0 AND iReadIndex <= MM_MAX_NUMBER_OF_CELL_ELEMENTS) THEN
			// Build remote symbol name
			sPrefix := CONCAT(sObjectIDentifier, '.stTrackStatus');
			// Data pointer
			pReadNodeData := ADR(aReadCellData.stCell);
			// Header data
			cbDataTotal := SIZEOF(aReadCellData.stCell);
			
			// Specify nodes to read by variable name
			sTrackServerSymbol := CONCAT(sPrefix, '.aCells[');
			sTrackServerSymbol := CONCAT(sTrackServerSymbol, UINT_TO_STRING(iReadIndex));
			sTrackServerSymbol := CONCAT(sTrackServerSymbol, ']');
			bReturn := TRUE;

			// continue to next type after this read!
			iReadIndex := 0;
			bReadDecPointVehicle := TRUE;	// Force reading of the vehicle at decision point before other vehicles
			IF (NOT bReadDecPointCellDone) THEN
				bReadDecPointCell := TRUE;
			END_IF
			eReadType := E_OPC_NodeType.Vehicles;
		ELSE
			// Read next type
			iReadIndex := 0;
			bReadDecPointVehicle := TRUE;	// Force reading of the vehicle at decision point before other vehicles
			eReadType := E_OPC_NodeType.Vehicles;
			bReturn := FALSE;
		END_IF

END_CASE

M_InitNodeData_ADS := bReturn;
END_METHOD

METHOD PROTECTED M_InitNodeData_OPCUA : BOOL
VAR
	i		: UINT;
	sPrefix : STRING;
END_VAR
VAR
	cbDataTotal2 : UINT;
END_VAR
// NOTE!!!
// Maximum of 10 elements to read for each Node List reading!


(* Node data, init to use string identifier and set namespace index *)
FOR i:=1 TO nMaxNodeIDsInList BY 1 DO
	aNodeIDs[i].eIdentifierType := eUAIdentifierType_String;
	aNodeIDs[i].nNamespaceIndex := nNameSpaceIndexNodes;
END_FOR

nNoOfNodes := 0;
cbDataTotal := 0;

// TEST
eReadType := E_OPC_NodeType.Nodes;
iReadIndex := 1;

// Comm type selection
CASE eReadType OF
	E_OPC_NodeType.Vehicles:
		// Limit number of elements
		iReadIndex := LIMIT(1, iReadIndex, MM_MAX_NUMBER_OF_VEHICLE_ELEMENTS);
		// Build remote symbol name
		sPrefix := CONCAT(sObjectIDentifier, '.stTrackStatus.aVehicles[');
		sPrefix := CONCAT(sPrefix, UINT_TO_STRING(iReadIndex));
		sPrefix := CONCAT(sPrefix, ']');
		// Data pointer
		pReadNodeData := ADR(aReadVehicleData[iReadIndex]);
		// Header data
		cbDataTotal := SIZEOF(aReadVehicleData[iReadIndex].stReadListReturnInfo);
		
		// Specify nodes to read by variable name
		nNoOfNodes := nNoOfNodes + 1;
		aNodeIDs[nNoOfNodes].sIdentifier := CONCAT(sPrefix, '.nVehicleID');
		acbDatas[nNoOfNodes] := SIZEOF(aReadVehicleData[iReadIndex].nVehicleID);
		cbDataTotal := cbDataTotal + acbDatas[nNoOfNodes];
		
		nNoOfNodes := nNoOfNodes + 1;
		aNodeIDs[nNoOfNodes].sIdentifier := CONCAT(sPrefix, '.bVehiclePresent');
		acbDatas[nNoOfNodes] := SIZEOF(aReadVehicleData[iReadIndex].bVehiclePresent);
		cbDataTotal := cbDataTotal + acbDatas[nNoOfNodes];
		
		nNoOfNodes := nNoOfNodes + 1;
		aNodeIDs[nNoOfNodes].sIdentifier := CONCAT(sPrefix, '.nState');
		acbDatas[nNoOfNodes] := SIZEOF(aReadVehicleData[iReadIndex].nState);
		cbDataTotal := cbDataTotal + acbDatas[nNoOfNodes];
		
		nNoOfNodes := nNoOfNodes + 1;
		aNodeIDs[nNoOfNodes].sIdentifier := CONCAT(sPrefix, '.nPathID');
		acbDatas[nNoOfNodes] := SIZEOF(aReadVehicleData[iReadIndex].nPathID);
		cbDataTotal := cbDataTotal + acbDatas[nNoOfNodes];
		
		nNoOfNodes := nNoOfNodes + 1;
		aNodeIDs[nNoOfNodes].sIdentifier := CONCAT(sPrefix, '.fPosition');
		acbDatas[nNoOfNodes] := SIZEOF(aReadVehicleData[iReadIndex].fPosition);
		cbDataTotal := cbDataTotal + acbDatas[nNoOfNodes];
		
		nNoOfNodes := nNoOfNodes + 1;
		aNodeIDs[nNoOfNodes].sIdentifier := CONCAT(sPrefix, '.nTargetPathID');
		acbDatas[nNoOfNodes] := SIZEOF(aReadVehicleData[iReadIndex].nTargetPathID);
		cbDataTotal := cbDataTotal + acbDatas[nNoOfNodes];
		
		nNoOfNodes := nNoOfNodes + 1;
		aNodeIDs[nNoOfNodes].sIdentifier := CONCAT(sPrefix, '.fTargetPosition');
		acbDatas[nNoOfNodes] := SIZEOF(aReadVehicleData[iReadIndex].fTargetPosition);
		cbDataTotal := cbDataTotal + acbDatas[nNoOfNodes];
		
		nNoOfNodes := nNoOfNodes + 1;
		aNodeIDs[nNoOfNodes].sIdentifier := CONCAT(sPrefix, '.fVelocity');
		acbDatas[nNoOfNodes] := SIZEOF(aReadVehicleData[iReadIndex].fVelocity);
		cbDataTotal := cbDataTotal + acbDatas[nNoOfNodes];
				
		// Read next vehicle value
		iReadIndex := iReadIndex+1;;
		IF (iReadIndex > MM_MAX_NUMBER_OF_VEHICLE_ELEMENTS) THEN
			// Read next type
			iReadIndex := 0;
			eReadType := E_OPC_NodeType.Paths;
		END_IF

	E_OPC_NodeType.Paths:
		// Limit number of elements
		iReadIndex := LIMIT(1, iReadIndex, MM_MAX_NUMBER_OF_PATH_ELEMENTS);
		// Build remote symbol name
		sPrefix := CONCAT(sObjectIDentifier, '.stTrackStatus.aPaths[');
		sPrefix := CONCAT(sPrefix, UINT_TO_STRING(iReadIndex));
		sPrefix := CONCAT(sPrefix, ']');
		// Data pointer
		pReadNodeData := ADR(aReadPathData[iReadIndex]);
		
		// Header data
		cbDataTotal := SIZEOF(aReadPathData[iReadIndex].stReadListReturnInfo);
		
		// Specify nodes to read by variable name
		nNoOfNodes := nNoOfNodes + 1;
		aNodeIDs[nNoOfNodes].sIdentifier := CONCAT(sPrefix, '.nPathID');
		acbDatas[nNoOfNodes] := SIZEOF(aReadPathData[iReadIndex].nPathID);
		cbDataTotal := cbDataTotal + acbDatas[nNoOfNodes];

		nNoOfNodes := nNoOfNodes + 1;
		aNodeIDs[nNoOfNodes].sIdentifier := CONCAT(sPrefix, '.sCellID');
		acbDatas[nNoOfNodes] := SIZEOF(aReadPathData[iReadIndex].sCellID);
		cbDataTotal := cbDataTotal + acbDatas[nNoOfNodes];

		nNoOfNodes := nNoOfNodes + 1;
		aNodeIDs[nNoOfNodes].sIdentifier := CONCAT(sPrefix, '.bPathPresent');
		acbDatas[nNoOfNodes] := SIZEOF(aReadPathData[iReadIndex].bPathPresent);
		cbDataTotal := cbDataTotal + acbDatas[nNoOfNodes];

		nNoOfNodes := nNoOfNodes + 1;
		aNodeIDs[nNoOfNodes].sIdentifier := CONCAT(sPrefix, '.nState');
		acbDatas[nNoOfNodes] := SIZEOF(aReadPathData[iReadIndex].nState);
		cbDataTotal := cbDataTotal + acbDatas[nNoOfNodes];

		// Read next path value
		iReadIndex := iReadIndex+1;
		IF (iReadIndex > MM_MAX_NUMBER_OF_PATH_ELEMENTS) THEN
			// Read next type
			iReadIndex := 0;
			eReadType := E_OPC_NodeType.Nodes;
			//eReadType := E_OPC_NodeType.Vehicles;
		END_IF
		
		
	E_OPC_NodeType.Nodes:
		// Limit number of elements
		iReadIndex := LIMIT(1, iReadIndex, 10);
		// Build remote symbol name
		sPrefix := CONCAT(sObjectIDentifier, '.stTrackStatus');
		// Data pointer
		pReadNodeData := ADR(aReadNodeData[iReadIndex]);
		
		// Header data
		cbDataTotal := SIZEOF(aReadNodeData[iReadIndex].stReadListReturnInfo);
		cbDataTotal2 := SIZEOF(aReadNodeData[iReadIndex]);
		
		// Specify nodes to read by variable name
		nNoOfNodes := nNoOfNodes + 1;
		aNodeIDs[nNoOfNodes].sIdentifier := CONCAT(sPrefix, '.aNodes[');
		aNodeIDs[nNoOfNodes].sIdentifier := CONCAT(aNodeIDs[nNoOfNodes].sIdentifier, UINT_TO_STRING(iReadIndex));
		aNodeIDs[nNoOfNodes].sIdentifier := CONCAT(aNodeIDs[nNoOfNodes].sIdentifier, ']');
		acbDatas[nNoOfNodes] := SIZEOF(aReadNodeData[iReadIndex].stNodeData);
		cbDataTotal := cbDataTotal + acbDatas[nNoOfNodes];

		// Read next node value
		iReadIndex := iReadIndex+1;
		IF (iReadIndex > 10) THEN
			// Read next type
			iReadIndex := 0;
			eReadType := E_OPC_NodeType.Vehicles;
		END_IF

END_CASE
END_METHOD

METHOD PROTECTED M_MappingData
VAR_INPUT
END_VAR
VAR
	i			: USINT;
	iRes		: UINT;
END_VAR
// Handle the mapping data from OPC UA (stCommand)

CASE eMappingDataState OF
	// Init state
	E_MappingDataState.Undefined:
		eMappingDataState := E_MappingDataState.CheckRequest;
	
	// Check command data request
	E_MappingDataState.CheckRequest:
		IF ((stMappingIn.ChangeRequest <> stMappingOut.ChangeStatus) AND (stMappingIn.ChangeRequest > 0)) THEN
			// Check if changes is allowed on mapping data (from LC)
			IF (stAdditionalDataIn.MESHandShakes.DataChangeStatusTransportMapping = stMappingOut.DataChange) THEN
				stMappingOut.ChangeAcknowlegde := stMappingIn.ChangeRequest;
				stMappingOut.DataChange := stMappingOut.DataChange + 1;
				
				// Find vehicle ID with specified carrier ID
				iMappingDataVehicleID := M_CarrierIDToVehicleID(stMappingIn.Carrier.CarrierID);
	
				// Check vehicle number
				IF (iMappingDataVehicleID > 0) THEN
					eMappingDataState := E_MappingDataState.UpdateMappingData;
				ELSE
					eMappingDataState := E_MappingDataState.Error;
				END_IF
			END_IF	
		END_IF	
	
	// Perform data update
	E_MappingDataState.UpdateMappingData:
		iRes := M_CallUpdateVehicleMappingData(	nVehicleID := iMappingDataVehicleID,
												sCarrierID := stMappingIn.Carrier.CarrierID, 
												bTool := stMappingIn.Carrier.Tool, 
												sToolID := stMappingIn.Carrier.ToolID, 
												bMaterial := stMappingIn.Carrier.Material,
												sMaterialID := stMappingIn.Carrier.MaterialID 	);
		IF (iRes = 2) THEN
			// Success.
			eMappingDataState := E_MappingDataState.UpdateReworkData;
		ELSIF (iRes = 3) THEN
			// Error!
			eMappingDataState := E_MappingDataState.Error;
		END_IF
	
	// Perform rework update
	E_MappingDataState.UpdateReworkData:
		iRes := M_CallUpdateVehicleReworkData(	nVehicleID := iMappingDataVehicleID,
												sCarrierID := stMappingIn.Carrier.CarrierID,
												bNOK := stMappingIn.Carrier.NOK	); 
		IF (iRes = 2) THEN
			// Success..
			eMappingDataState := E_MappingDataState.Done;
		ELSIF (iRes = 3) THEN
			// Error!
			eMappingDataState := E_MappingDataState.Error;
		END_IF
	
	E_MappingDataState.Done:
		// Completed... Update output mapping data
		stMappingOut.ValidRequest := TRUE;
		stMappingOut.Carrier := stMappingIn.Carrier;
		stMappingOut.StationBuffer := stMappingIn.StationBuffer;
		stMappingOut.ChangeStatus := stMappingIn.ChangeRequest;
		stMappingOut.DataChange := stMappingOut.DataChange + 1;
		eMappingDataState := E_MappingDataState.Undefined;
	
	E_MappingDataState.Error:
		// Error... Valid request = FALSE
		stMappingOut.ValidRequest := FALSE;
		stMappingOut.ChangeStatus := stMappingIn.ChangeRequest;
		stMappingOut.DataChange := stMappingOut.DataChange + 1;
		eMappingDataState := E_MappingDataState.Undefined;
	
END_CASE
END_METHOD

METHOD PROTECTED M_ReworkData
VAR_INPUT
END_VAR
VAR
	i			: USINT;
	iRes		: UINT;
END_VAR
// Handle the mapping data from OPC UA (stCommand)

CASE eReworkDataState OF
	// Init state
	E_ReworkDataState.Undefined:
		bReworkValue := FALSE;
		iReworkDataStation := 0;
		iReworkDataStationNo := 0;
		eReworkDataState := E_ReworkDataState.CheckRequest;
	
	// Check command data request
	E_ReworkDataState.CheckRequest:
		FOR i := 1 TO 5 BY 1 DO
			/////////////////////////////////////////////////////////////////////////////////////////////////////////////////////
			// Rework completed from station (shoe rework is done handled)
			/////////////////////////////////////////////////////////////////////////////////////////////////////////////////////
			IF (abStation1ReworkDone[i]) THEN
				iReworkDataStation := i;
				iReworkDataStationNo := 1;

				// Check vehicle at station
				iReworkDataVehicleID := aStations[iReworkDataStation].stStationData1.nCurrentVehicleID;
				IF ((iReworkDataVehicleID > 0) AND (iReworkDataVehicleID <= MM_MAX_NUMBER_OF_VEHICLE_ELEMENTS) ) THEN
					// There is a vehicle on that station! Get the Carrier ID
					sReworkDataCarrierID := aReadVehicleData[iReworkDataVehicleID].stVehicle.sCarrierID;
					
					// Check carrier ID of vehicle
					IF (sReworkDataCarrierID <> '') THEN
						bReworkValue := FALSE;	// Set carrier status to rework NOT needed!
						eReworkDataState := E_ReworkDataState.UpdateReworkData;
					ELSE
						// Error!
						eReworkDataState := E_ReworkDataState.Error;
					
					END_IF
				ELSE
					// Error!
					eReworkDataState := E_ReworkDataState.Error;
				
				END_IF

				EXIT;
				
			ELSIF (abStation2ReworkDone[i]) THEN
				iReworkDataStation := i;
				iReworkDataStationNo := 2;

				iReworkDataVehicleID := aStations[iReworkDataStation].stStationData2.nCurrentVehicleID;
				IF ((iReworkDataVehicleID > 0) AND (iReworkDataVehicleID <= MM_MAX_NUMBER_OF_VEHICLE_ELEMENTS) ) THEN
					// There is a vehicle on that station! Get the Carrier ID
					sReworkDataCarrierID := aReadVehicleData[iReworkDataVehicleID].stVehicle.sCarrierID;
					
					// Check carrier ID of vehicle
					IF (sReworkDataCarrierID <> '') THEN
						bReworkValue := FALSE;	// Set carrier status to rework NOT needed!
						eReworkDataState := E_ReworkDataState.UpdateReworkData;
					ELSE
						// Error!
						eReworkDataState := E_ReworkDataState.Error;
					
					END_IF				
				ELSE
					// Error!
					eReworkDataState := E_ReworkDataState.Error;
				
				END_IF

				EXIT;

			/////////////////////////////////////////////////////////////////////////////////////////////////////////////////////
			// Rework request from station (shoe needs to be reworked)
			/////////////////////////////////////////////////////////////////////////////////////////////////////////////////////
			ELSIF (abStation1ReworkReq[i]) THEN
				iReworkDataStation := i;
				iReworkDataStationNo := 1;

				// Check vehicle at station
				iReworkDataVehicleID := aStations[iReworkDataStation].stStationData1.nCurrentVehicleID;
				IF ((iReworkDataVehicleID > 0) AND (iReworkDataVehicleID <= MM_MAX_NUMBER_OF_VEHICLE_ELEMENTS) ) THEN
					// There is a vehicle on that station! Get the Carrier ID
					sReworkDataCarrierID := aReadVehicleData[iReworkDataVehicleID].stVehicle.sCarrierID;
					
					// Check carrier ID of vehicle
					IF (sReworkDataCarrierID <> '') THEN
						bReworkValue := TRUE;	// Set carrier status to rework needed!
						eReworkDataState := E_ReworkDataState.UpdateReworkData;
					ELSE
						// Error!
						eReworkDataState := E_ReworkDataState.Error;
					
					END_IF
				ELSE
					// Error!
					eReworkDataState := E_ReworkDataState.Error;
				
				END_IF

				EXIT;
				
			ELSIF (abStation2ReworkReq[i]) THEN
				iReworkDataStation := i;
				iReworkDataStationNo := 2;

				iReworkDataVehicleID := aStations[iReworkDataStation].stStationData2.nCurrentVehicleID;
				IF ((iReworkDataVehicleID > 0) AND (iReworkDataVehicleID <= MM_MAX_NUMBER_OF_VEHICLE_ELEMENTS) ) THEN
					// There is a vehicle on that station! Get the Carrier ID
					sReworkDataCarrierID := aReadVehicleData[iReworkDataVehicleID].stVehicle.sCarrierID;
					
					// Check carrier ID of vehicle
					IF (sReworkDataCarrierID <> '') THEN
						bReworkValue := TRUE;	// Set carrier status to rework needed!
						eReworkDataState := E_ReworkDataState.UpdateReworkData;
					ELSE
						// Error!
						eReworkDataState := E_ReworkDataState.Error;
					
					END_IF				
				ELSE
					// Error!
					eReworkDataState := E_ReworkDataState.Error;
				
				END_IF

				EXIT;
			END_IF
		END_FOR
	
	// Perform rework update
	E_ReworkDataState.UpdateReworkData:
		iRes := M_CallUpdateVehicleReworkData(	nVehicleID := iReworkDataVehicleID,
												sCarrierID := sReworkDataCarrierID,
												bNOK := bReworkValue 	);
		IF (iRes = 2) THEN
			// Success..
			F_LogLine(CONCAT('TC_RWK: Vehicle ', CONCAT(UINT_TO_STRING(iReworkDataVehicleID), ' NOK set to %d')), BOOL_TO_DINT(bReworkValue));
			eReworkDataState := E_ReworkDataState.Done;
		ELSIF (iRes = 3) THEN
			// Error!
			eReworkDataState := E_ReworkDataState.Error;
		END_IF
	
	E_ReworkDataState.Done:
		// Completed... Wait until activation bit is sert to FALSE (when vehicle has been removed from station)
		IF (bReworkValue) THEN
			IF (iReworkDataStationNo = 1) THEN
				IF (NOT abStation1ReworkReq[iReworkDataStation]) THEN
					eReworkDataState := E_ReworkDataState.Undefined;		
				END_IF
	
			ELSIF (iReworkDataStationNo = 2) THEN
				IF (NOT abStation2ReworkReq[iReworkDataStation]) THEN
					eReworkDataState := E_ReworkDataState.Undefined;
				END_IF
	
			END_IF
		ELSE
			IF (iReworkDataStationNo = 1) THEN
				IF (NOT abStation1ReworkDone[iReworkDataStation]) THEN
					eReworkDataState := E_ReworkDataState.Undefined;		
				END_IF
	
			ELSIF (iReworkDataStationNo = 2) THEN
				IF (NOT abStation2ReworkDone[iReworkDataStation]) THEN
					eReworkDataState := E_ReworkDataState.Undefined;
				END_IF
	
			END_IF
		END_IF
	
	E_ReworkDataState.Error:
		// Error... Wait until activation bit is sert to FALSE (when vehicle has been removed from station)
		// TODO!!! Alarm!
		IF (bReworkValue) THEN
			IF (iReworkDataStationNo = 1) THEN
				IF (NOT abStation1ReworkReq[iReworkDataStation]) THEN
					eReworkDataState := E_ReworkDataState.Undefined;		
				END_IF
	
			ELSIF (iReworkDataStationNo = 2) THEN
				IF (NOT abStation2ReworkReq[iReworkDataStation]) THEN
					eReworkDataState := E_ReworkDataState.Undefined;
				END_IF
	
			END_IF
		ELSE
			IF (iReworkDataStationNo = 1) THEN
				IF (NOT abStation1ReworkDone[iReworkDataStation]) THEN
					eReworkDataState := E_ReworkDataState.Undefined;		
				END_IF
	
			ELSIF (iReworkDataStationNo = 2) THEN
				IF (NOT abStation2ReworkDone[iReworkDataStation]) THEN
					eReworkDataState := E_ReworkDataState.Undefined;
				END_IF
	
			END_IF
		END_IF

END_CASE
END_METHOD

METHOD PROTECTED M_Run : BOOL
VAR_INPUT
END_VAR
VAR
	i	: USINT;
END_VAR
// Get system time
fbGetTime(	NETID:= '',	// Local PLC 
			START:= NOT fbGetTime.START AND NOT fbGetTime.BUSY, 
			TMOUT:= T#5S	);

///////////////////////////////////////////////////////////////////////////////////////////////////////////////////
// FB's for method calling
///////////////////////////////////////////////////////////////////////////////////////////////////////////////////
	(* Handle server connect *)
	fbConnectMethod(	Execute				:= , 
						ServerUrl			:= sTrackServerUrl, 
						SessionConnectInfo	:= stConnectInfoMethod, 
						Timeout				:= T#10S, 
						ConnectionHdl		=> , 
						Done				=> , 
						Busy				=> , 
						Error				=> , 
						ErrorID				=> 	);
					
	(* Handle server dicconnect *)
	fbDisconnectMethod(	Execute				:= , 
						ConnectionHdl		:= nConnectHdlMethod, 
						Timeout				:= T#10S, 
						Done				=> , 
						Busy				=> , 
						Error				=> , 
						ErrorID				=> 	);
						
	(* Get namepsace *)
	fbGetNamespaceMethod(	Execute				:= , 
							ConnectionHdl		:= nConnectHdlMethod, 
							NamespaceUri		:= sNameSpaceUri, 
							Timeout				:= T#10S, 
							NamespaceIndex		=> , 
							Done				=> , 
							Busy				=> , 
							Error				=> , 
							ErrorID				=> 	);
	
	(* Get method handle *)
	stObjectNodeID.nNamespaceIndex := nNameSpaceIndexMethod;
	stObjectNodeID.sIdentifier := sObjectIDentifier;
	stMethodNodeID.nNamespaceIndex := nNameSpaceIndexMethod;
	stMethodNodeID.sIdentifier := sMethodIdentifier;
	fbGetHandleMethod(	Execute				:= , 
						ConnectionHdl		:= nConnectHdlMethod, 
						ObjectNodeID		:= stObjectNodeID, 
						MethodNodeID		:= stMethodNodeID, 
						Timeout				:= T#10S, 
						MethodHdl			=> , 
						Done				=> , 
						Busy				=> , 
						Error				=> , 
						ErrorID				=>	);
	
	(* Call method *)
	fbCallMethod(	Execute					:= , 
					ConnectionHdl			:= nConnectHdlMethod, 
					MethodHdl				:= nHandleMethod, 
					nNumberOfInputArguments	:= , 
					pInputArgInfo			:= , 
					cbInputArgInfo			:= , 
					pInputArgData			:= , 
					cbInputArgData			:= , 
					pInputWriteData			:= 0,
					cbInputWriteData		:= 0,
					nNumberOfOutputArguments:= , 
					pOutputArgInfo			:= , 
					cbOutputArgInfo			:= , 
					pOutputArgInfoAndData	:= , 
					cbOutputArgInfoAndData	:= , 
					Timeout					:= T#10S, 
					cbRead_R				=> , 
					Done					=> , 
					Busy					=> , 
					Error					=> , 
					ErrorID					=> );
	
	(* Release method handle *)
	fbReleaseHandleMethod(	Execute			:= , 
							ConnectionHdl	:= nConnectHdlMethod, 
							MethodHdl		:= nHandleMethod, 
							Timeout			:= T#10S, 
							Done			=> , 
							Busy			=> , 
							Error			=> , 
							ErrorID			=> 	);

///////////////////////////////////////////////////////////////////////////////////////////////////////////////////
// FB's for method calling
///////////////////////////////////////////////////////////////////////////////////////////////////////////////////
	(* Handle server connect *)
	fbConnectNodes(	Execute				:= , 
					ServerUrl			:= sTrackServerUrl, 
					SessionConnectInfo	:= stConnectInfoNodes, 
					Timeout				:= T#10S, 
					ConnectionHdl		=> , 
					Done				=> , 
					Busy				=> , 
					Error				=> , 
					ErrorID				=> 	);
					
	(* Handle server dicconnect *)
	fbDisconnectNodes(	Execute				:= , 
						ConnectionHdl		:= nConnectHandleNodes, 
						Timeout				:= T#10S, 
						Done				=> , 
						Busy				=> , 
						Error				=> , 
						ErrorID				=> 	);
						
	(* Get namepsace *)
	fbGetNamespaceNodes(	Execute				:= , 
						ConnectionHdl		:= nConnectHandleNodes, 
						NamespaceUri		:= sNameSpaceUri, 
						Timeout				:= T#10S, 
						NamespaceIndex		=> , 
						Done				=> , 
						Busy				=> , 
						Error				=> , 
						ErrorID				=> 	);
	
	(* Get node handle *)
	fbGetHandleNodes(	Execute				:= , 
						ConnectionHdl		:= nConnectHandleNodes, 
						NodeIDCount			:= nNoOfNodes,
						NodeIDs				:= aNodeIDs, 
						Timeout				:= T#10S, 
						NodeHdls			=> , 
						Done				=> , 
						Busy				=> , 
						Error				=> , 
						ErrorID				=> 	);
		
	(* Read node data *)
	fbReadNodes(	Execute:= , 
					ConnectionHdl			:= nConnectHandleNodes,
					NodeHdlCount			:= nNoOfNodes,
					NodeHdls				:= anHandleNodes, 
					stNodeAddInfo			:= astNodeAddInfo, 
					pVariable				:= pReadNodeData, 
					cbData					:= acbDatas,
					cbDataTotal				:= cbDataTotal, 
					Timeout					:= T#10S, 
					Done					=> , 
					Busy					=> , 
					Error					=> , 
					ErrorID					=> , 
					cbData_R				=> 	);
					
	(* Release node handle list *)
	fbReleaseHandleNodes(	Execute			:= , 
							ConnectionHdl	:= nConnectHandleNodes, 
							NodeHdlCount	:= nNoOfNodes, 
							NodeHdls		:= anHandleNodes, 
							Timeout			:= T#10S, 
							NodeErrorIDs	=> , 
							Done			=> , 
							Busy			=> , 
							Error			=> , 
							ErrorID			=> 	);
	
	(* Read interval *)
	tonReadInterval(	IN	:= ,
						PT	:= REAL_TO_TIME(rReadInterval * 1000.0),
						Q	=> ,
						ET	=> 	);
						
	(* Error automatic reset delay *)
	tonErrorReset(		IN	:= ,
						PT	:= REAL_TO_TIME(rErrorResetDelay * 1000.0),
						Q	=> ,
						ET	=> 	);

// Update Additional Data variables
	stAdditionaldataOut.bConnectedMethod := bConnectedMethod;
	stAdditionaldataOut.bConnectedNode := bConnectedNode;
	stAdditionaldataOut.bTrackReady := P_bTrackReady;
END_METHOD

METHOD PROTECTED M_StateMachine : BOOL
VAR_INPUT
END_VAR
VAR
	iRes	: INT;
	i		: UINT;
END_VAR

CASE eTrackState OF
	E_TrackState.Undefined:
		bStarted := FALSE;
		bSuspended := FALSE;
		iStationID := 1;
		iPathID := 1;
		iPathIndex := 1;
		IF (bConnectedMethod AND bConnectedNode) THEN
			// Communication connections established
			IF (bEnable) THEN
				eTrackState := E_TrackState.CheckInitDone;
			END_IF
		END_IF
	
	E_TrackState.CheckInitDone:
		// Check if track has been setup from this cell already on the track server
		iRes := M_CallGetCellIndex(sCellID);
		IF (iRes = 2) THEN
			// Success... Init done
			// Save found index
			iThisCellIndex := stGetCellIndexData.stOutput.nCellIndex;
			IF (iThisCellIndex > 0) THEN
				bTrackInitDone := TRUE;
				eTrackState := E_TrackState.Starting;
			ELSE
				bTrackInitDone := FALSE;
				bStationData1Done := FALSE;
				bStationData2Done := FALSE;
				// Clear station index
				FOR i := 1 TO 5 BY 1 DO
					iThisStationIndex[i] := 0;
				END_FOR
				eTrackState := E_TrackState.WaitAllowInit;
			END_IF
		ELSIF (iRes = 3) THEN
			// Error!
			// Clear station index
			FOR i := 1 TO 5 BY 1 DO
				iThisStationIndex[i] := 0;
			END_FOR
			eTrackState := E_TrackState.WaitAllowInit;
		END_IF
	
//	E_TrackState.InitDecisionPoint:
//		// Initialized with stations
//		eTrackState := E_TrackState.InitStations;
	
	E_TrackState.WaitAllowInit:
		// Initialized with stations
		IF (stAdditionalDataIn.bAllowInit) THEN
			stAdditionalDataIn.bAllowInit := FALSE;
			eTrackState := E_TrackState.InitStations;
		ELSIF (NOT bEnable OR NOT bConnectedMethod OR NOT bConnectedNode) THEN
			eTrackState := E_TrackState.Undefined;
		END_IF

	E_TrackState.InitStations:
		IF (aStations[iStationID].bPresent) THEN
			IF (aStations[iStationID].stStationData2.stLocation.nPathID > 0) THEN
				// Double position station
				iRes := M_CallAddStationDouble(nStationNo := iStationID);
				IF (iRes = 2) THEN
					// Success... Next station
					iStationID := iStationID + 1;
				ELSIF (iRes = 3) THEN
					// Error!
					// TODO!!!
					;				
				END_IF
			ELSE
				// Single position station
				iRes := M_CallAddStationSingle(nStationNo := iStationID);
				IF (iRes = 2) THEN
					// Success... Next station
					iStationID := iStationID + 1;
				ELSIF (iRes = 3) THEN
					// Error!
					// TODO!!!
					;				
				END_IF
			END_IF
		ELSE
			// Not enabled... Next station
			iStationID := iStationID + 1;
		END_IF
		IF (iStationID >= 5) THEN
			// All added
			iStationID := 1;
//			eTrackState := E_TrackState.InitPathsStations;	// init paths from stations, traffic lights and decision point 
			eTrackState := E_TrackState.SetPreBufferAdjust;
		END_IF
		
	E_TrackState.SetPreBufferAdjust:
		IF (aStations[iStationID].bPresent) THEN
			IF (aStationPreBufAdj[iStationID] <> 0.0) THEN
				iRes := M_CallAdjustBufferPosition(	nStationNo := iStationID,
													eBufferType := E_MMStationBuffer.eMMStationBuffer_PreProcess,
													rDistance := aStationPreBufAdj[iStationID]	);
				IF (iRes = 2) THEN
					// Success... Next station
					iStationID := iStationID + 1;
				ELSIF (iRes = 3) THEN
					// Error!
					// TODO!!!
					;
				END_IF
				
			ELSE
				// No adustment needed
				iStationID := iStationID + 1;
			END_IF
		ELSE
			// Not enabled... Next station
			iStationID := iStationID + 1;
		END_IF
		IF (iStationID >= 5) THEN
			// All checked/adjusted
			iStationID := 1;
			eTrackState := E_TrackState.SetPostBufferAdjust;
		END_IF
		
	E_TrackState.SetPostBufferAdjust:
		IF (aStations[iStationID].bPresent) THEN
			IF (aStationPostBufAdj[iStationID] <> 0.0) THEN
				iRes := M_CallAdjustBufferPosition(	nStationNo := iStationID,
													eBufferType := E_MMStationBuffer.eMMStationBuffer_PostProcess,
													rDistance := aStationPostBufAdj[iStationID]	);
				IF (iRes = 2) THEN
					// Success... Next station
					iStationID := iStationID + 1;
				ELSIF (iRes = 3) THEN
					// Error!
					// TODO!!!
					;
				END_IF
				
			ELSE
				// No adustment needed
				iStationID := iStationID + 1;
			END_IF
		ELSE
			// Not enabled... Next station
			iStationID := iStationID + 1;
		END_IF
		IF (iStationID >= 5) THEN
			// All checked/adjusted
			iStationID := 1;
			eTrackState := E_TrackState.InitPaths;
		END_IF
		
	// Create/init paths on track server for this cell
	E_TrackState.InitPaths:	
		IF (aPaths[iPathID] > 0) THEN
			iRes := M_CallAddPath(nPathNo := aPaths[iPathID]);
			IF (iRes = 2) THEN
				// Success... Next Path
				abControlledPaths[aPaths[iPathID]] := TRUE;
				iPathID := iPathID + 1;
			ELSIF (iRes = 3) THEN
				// Error!
				// TODO!!!
				;
			END_IF
		ELSE
			// All added
			iPathID := 1;
			eTrackState := E_TrackState.InitGetCellIndex;
		END_IF
(*		
	// Create/init paths on track server for this cell
	E_TrackState.InitPathsStations:	
		IF (aStations[iStationID].bPresent) THEN
			IF (NOT bStationData1Done) THEN
				iRes := M_CallAddPath(nPathNo := aStations[iStationID].stStationData1.stLocation.nPathID);
				IF (iRes = 2) THEN
					// Success... Next station
					abControlledPaths[aStations[iStationID].stStationData1.stLocation.nPathID] := TRUE;
					bStationData1Done := TRUE;
					IF (aStations[iStationID].stStationData1.stLocation.nPathID = aStations[iStationID].stStationData2.stLocation.nPathID) THEN
						// Station 2 is on the same path
						bStationData2Done := TRUE;
						iStationID := iStationID + 1;						
					ELSE
						// Station 2 is on a different path
						
					END_IF
				ELSIF (iRes = 3) THEN
					// Error!
					// TODO!!!
					;
				END_IF
			ELSIF (NOT bStationData2Done) THEN
				iRes := M_CallAddPath(nPathNo := aStations[iStationID].stStationData2.stLocation.nPathID);
				IF (iRes = 2) THEN
					// Success... Next station
					abControlledPaths[aStations[iStationID].stStationData2.stLocation.nPathID] := TRUE;
					bStationData2Done := TRUE;
					iStationID := iStationID + 1;
				ELSIF (iRes = 3) THEN
					// Error!
					// TODO!!!
					;
				END_IF
			END_IF
		ELSE
			// Not enabled... Next station
			iStationID := iStationID + 1;
		END_IF
		IF (iStationID >= 5) THEN
			// All added
			iStationID := 1;
			eTrackState := E_TrackState.InitPathsDecisionPoint;
		END_IF
	
	// Create/init paths on track server for this cell
	E_TrackState.InitPathsDecisionPoint:	
		IF (aStations[iStationID].bPresent) THEN
			iRes := M_CallAddPath(nPathNo := aStations[iStationID].stDecisionLocation.nPathID);
			IF (iRes = 2) THEN
				// Success... Next station
				abControlledPaths[aStations[iStationID].stDecisionLocation.nPathID] := TRUE;
				iStationID := iStationID + 1;
			ELSIF (iRes = 3) THEN
				// Error!
				// TODO!!!
				;
			END_IF
		ELSE
			// Not enabled... Next station
			iStationID := iStationID + 1;
		END_IF
		IF (iStationID >= 5) THEN
			// All added
			iStationID := 1;
			eTrackState := E_TrackState.InitPathsTrafficLight;
		END_IF

	// Create/init paths on track server for this cell
	E_TrackState.InitPathsTrafficLight:	
		IF (stTrafficLightLocation.nPathID > 0) THEN
			iRes := M_CallAddPath(nPathNo := stTrafficLightLocation.nPathID);	
			IF (iRes = 2) THEN
				// Success
				abControlledPaths[stTrafficLightLocation.nPathID] := TRUE;
				eTrackState := E_TrackState.InitGetCellIndex;
			ELSIF (iRes = 3) THEN
				// Error!
				// TODO!!!
				;
			END_IF
		ELSE
			eTrackState := E_TrackState.InitGetCellIndex;			
		END_IF
*)
	E_TrackState.InitGetCellIndex:
		iRes := M_CallGetCellIndex(sCellID);
		IF (iRes = 2) THEN
			// Success... Init done
			// Save found index
			iThisCellIndex := stGetCellIndexData.stOutput.nCellIndex;
			bTrackInitDone := TRUE;
			eTrackState := E_TrackState.Resetting;
		ELSIF (iRes = 3) THEN
			// Error!
			// TODO!!!
			;
		END_IF	
	
	E_TrackState.Starting:
		IF (abControlledPaths[iPathID]) THEN
			// This path is controlled by this cell
			iRes := M_CallStartPath(nPathNo := iPathID);
			IF (iRes = 2) THEN
				// Success... Next station
				iPathID := iPathID + 1;
			ELSIF (iRes = 3) THEN
				// Error!
				// TODO!!!
				;
			END_IF
			
		ELSE
			iPathID := iPathID + 1;
		END_IF
		IF (iPathID >= MM_MAX_NUMBER_OF_PATH_ELEMENTS) THEN
			// All started
			iPathID := 1;
			bPathsOperational := TRUE;
			bPathsSuspended := FALSE;
			eTrackState := E_TrackState.StartCheck;
		END_IF
	
	E_TrackState.StartCheck:
		IF (abControlledPaths[iPathID]) THEN
			// Is this path controlled by this cell
			IF (aReadPathData[iPathID].stPathData.bPathPresent AND (aReadPathData[iPathID].stPathData.nState = E_MMPathState.eMMPathState_Operational)) THEN
				// This path is operational
				bPathsOperational := bPathsOperational AND TRUE;
			ELSE
				// Not operational
				bPathsOperational := FALSE;
			END_IF
			IF (aReadPathData[iPathID].stPathData.nMotionStatus = E_MMPathMotionStatus.eMMPathMotionStatus_SuspendedByCommand) THEN
				// This path is suspended!
				bPathsSuspended := TRUE;
			END_IF
		END_IF
		iPathID := iPathID + 1;
		IF (iPathID > MM_MAX_NUMBER_OF_PATH_ELEMENTS) THEN
			IF (bPathsOperational) THEN
				// All paths OK... Continue
				iPathID := 1;
				eTrackState := E_TrackState.InitTrafficLight;
			ELSIF (NOT bEnable) THEN
				// Stop
				eTrackState := E_TrackState.Undefined;			
			ELSE
				// All paths NOT OK!
				bPathsOperational := TRUE;
				bPathsSuspended := FALSE;
				iPathID := 1;
			END_IF
		END_IF
	
	E_TrackState.InitTrafficLight:
		// Check if Traffic light is defined!
		IF (stTrafficLightLocation.nPathID > 0) THEN
			iRes := M_CallAddTrafficLight(	nTrafficLightID := 1,
											nPathID := stTrafficLightLocation.nPathID,
											fPosition := stTrafficLightLocation.fPosition);
			IF (iRes = 2) THEN
				// Success... Init done
				eTrackState := E_TrackState.InitTrafficLight2;
			ELSIF (iRes = 3) THEN
				// Error!
				// TODO!!!
				;				
			END_IF
		ELSE
			eTrackState := E_TrackState.InitTrafficLight2;
		END_IF
	
	E_TrackState.InitTrafficLight2:
		// Check if Traffic light 2 is defined!
		IF (stTrafficLight2Location.nPathID > 0) THEN
			iRes := M_CallAddTrafficLight(	nTrafficLightID := 2,
											nPathID := stTrafficLight2Location.nPathID,
											fPosition := stTrafficLight2Location.fPosition);
			IF (iRes = 2) THEN
				// Success... Init done
				eTrackState := E_TrackState.InitPathSegment;
			ELSIF (iRes = 3) THEN
				// Error!
				// TODO!!!
				;				
			END_IF
		ELSE
			eTrackState := E_TrackState.InitPathSegment;
		END_IF

	E_TrackState.InitPathSegment:
		// Check if Path Segment is defined!
		IF (stExitPointSeg1LocBegin.nPathID > 0) THEN
			iRes := M_CallAddPathSegment(	iSegmentNo := 1,
											nPathNo := stExitPointSeg1LocBegin.nPathID,
											rBeginPosition := stExitPointSeg1LocBegin.fPosition,
											rEndPosition := stExitPointSeg1LocEnd.fPosition);
			IF (iRes = 2) THEN
				// Success... Init done
				eTrackState := E_TrackState.InitPathSegment2;
			ELSIF (iRes = 3) THEN
				// Error!
				// TODO!!!
				;				
			END_IF
		ELSE
			eTrackState := E_TrackState.InitPathSegment2;
		END_IF
	
	E_TrackState.InitPathSegment2:
		// Check if Path Segment is defined!
		IF (stExitPointSeg2LocBegin.nPathID > 0) THEN
			iRes := M_CallAddPathSegment(	iSegmentNo := 2,
											nPathNo := stExitPointSeg2LocBegin.nPathID,
											rBeginPosition := stExitPointSeg2LocBegin.fPosition,
											rEndPosition := stExitPointSeg2LocEnd.fPosition);
			IF (iRes = 2) THEN
				// Success... Init done
				eTrackState := E_TrackState.InitVehicles;
			ELSIF (iRes = 3) THEN
				// Error!
				// TODO!!!
				;				
			END_IF
		ELSE
			eTrackState := E_TrackState.InitVehicles;
		END_IF
	
	E_TrackState.InitVehicles:
		IF (bVehicleInitDone) THEN
			// Init done, go to started!
			eTrackState := E_TrackState.Started;
		ELSE
			iVehicleIndex := iVehicleIndex + 1;	// Start from 0!
			IF (aReadCellData.stCell.anVehicles[iVehicleIndex] > 0) THEN
				// Handle this vehicle
				iRes := M_CallMoveVehicleToScanner(	eInputType := E_MMVehicleInputType.eMMVehicleInputType_VehicleID,
													sInput := UINT_TO_STRING(aReadCellData.stCell.anVehicles[iVehicleIndex]),
													eDirection := E_MMDirection.eMMDirection_Forward, 
													fVelocity := 1,
													fAcceleration := 1 	);
				IF (iRes = 2) THEN
					// Next vehicle
					iVehicleIndex := iVehicleIndex + 1;
				ELSIF (iRes = 3) THEN
					// Error!
					// TODO!!!
					;
				END_IF
			ELSE
				// Next vehicle
				iVehicleIndex := iVehicleIndex + 1;
			END_IF
			IF (iVehicleIndex >= MM_MAX_NUMBER_OF_VEHICLE_ELEMENTS) THEN
				// All inited
				bVehicleInitDone := TRUE;
				iVehicleIndex := 0;
				eTrackState := E_TrackState.Started;
			END_IF
		END_IF
		
	E_TrackState.Started:
		bStarted := TRUE;
		IF (NOT bEnable) THEN
			// Disable
			eTrackState := E_TrackState.Undefined;
		ELSIF (iThisCellIndex <= 0) THEN
			// Re-Init cell index from track server
			iRes := M_CallGetCellIndex(sCellID);
			IF (iRes = 2) THEN
				// Success... Init done
				// Save found index
				iThisCellIndex := stGetCellIndexData.stOutput.nCellIndex;
			ELSIF (iRes = 3) THEN
				// Error!
				// TODO!!!
				;
			END_IF	
		ELSIF (bSuspend) THEN
			// Activate suspend on paths
			eTrackState := E_TrackState.Suspend;
		ELSIF (bPathsSuspended AND NOT bSuspend) THEN
			// Some paths are suspended and should not be
			eTrackState := E_TrackState.Resume;
		END_IF

	E_TrackState.Suspend:
		IF ( abControlledPaths[iPathID] AND (aReadPathData[iPathID].stPathData.nMotionStatus <> E_MMPathMotionStatus.eMMPathMotionStatus_SuspendedByCommand) ) THEN
			// This path is controlled by this cell and is not suspended
			iRes := M_CallSuspendPath(nPathNo := iPathID);
			IF (iRes = 2) THEN
				// Success... Next station
				iPathID := iPathID + 1;
			ELSIF (iRes = 3) THEN
				// Error!
				// TODO!!!
				;
			END_IF
		ELSE
			iPathID := iPathID + 1;
		END_IF
		IF (iPathID >= MM_MAX_NUMBER_OF_PATH_ELEMENTS) THEN
			// All suspended
			iPathID := 1;
			bPathsSuspended := TRUE;
			eTrackState := E_TrackState.Suspending;
		END_IF
		
	E_TrackState.Suspending:
		IF (abControlledPaths[iPathID]) THEN
			// Is this path controlled by this cell
			IF (aReadPathData[iPathID].stPathData.nMotionStatus = E_MMPathMotionStatus.eMMPathMotionStatus_SuspendedByCommand) THEN
				// This path is suspended
				bPathsSuspended := bPathsSuspended AND TRUE;
			ELSE
				// Not operational
				bPathsSuspended := FALSE;
			END_IF
		END_IF
		iPathID := iPathID + 1;
		IF (iPathID > MM_MAX_NUMBER_OF_PATH_ELEMENTS) THEN
			IF (bPathsSuspended) THEN
				// All paths Suspended... Continue
				iPathID := 1;
				eTrackState := E_TrackState.Suspended;
			ELSIF (NOT bEnable) THEN
				// Stop
				eTrackState := E_TrackState.Undefined;			
			ELSE
				// All paths NOT Suspended!
				iPathID := 1;
				bPathsSuspended := TRUE;
			END_IF
		END_IF		
	
	E_TrackState.Suspended:
		IF (NOT bSuspend) THEN
			bSuspended := FALSE;
			eTrackState := E_TrackState.Resume;
		ELSIF (NOT bEnable) THEN
			eTrackState := E_TrackState.Undefined;			
		END_IF
		
	E_TrackState.Resume:
		IF ( abControlledPaths[iPathID] AND aReadPathData[iPathID].stPathData.nMotionStatus = E_MMPathMotionStatus.eMMPathMotionStatus_SuspendedByCommand ) THEN
			// This path is controlled by this cell
			iRes := M_CallResumePath(nPathNo := iPathID);
			IF (iRes = 2) THEN
				// Success... Next station
				iPathID := iPathID + 1;
			ELSIF (iRes = 3) THEN
				// Error!
				// TODO!!!
				;
			END_IF
			
		ELSE
			iPathID := iPathID + 1;
		END_IF
		IF (iPathID >= MM_MAX_NUMBER_OF_PATH_ELEMENTS) THEN
			// All started
			iPathID := 1;
			bPathsResumed := TRUE;
			eTrackState := E_TrackState.Resuming;
		END_IF
	
	E_TrackState.Resuming:
		IF (abControlledPaths[iPathID]) THEN
			// Is this path controlled by this cell
			IF (aReadPathData[iPathID].stPathData.nMotionStatus <> E_MMPathMotionStatus.eMMPathMotionStatus_SuspendedByCommand) THEN
				// This path is operational
				bPathsResumed := bPathsResumed AND TRUE;
			ELSE
				// Not operational
				bPathsResumed := FALSE;
			END_IF
		END_IF
		iPathID := iPathID + 1;
		IF (iPathID > MM_MAX_NUMBER_OF_PATH_ELEMENTS) THEN
			IF (bPathsResumed) THEN
				// All paths Resumed... Continue
				iPathID := 1;
				bPathsSuspended := FALSE;
				eTrackState := E_TrackState.Started;
			ELSIF (NOT bEnable) THEN
				// Stop
				eTrackState := E_TrackState.Undefined;			
			ELSE
				// All paths NOT OK!
				bPathsResumed := TRUE;
				iPathID := 1;
			END_IF
		END_IF		
	
	E_TrackState.Resetting:
		IF (abControlledPaths[iPathID]) THEN
			// This path is controlled by this cell
			iRes := M_CallResetPath(nPathNo := iPathID);
			IF (iRes = 2) THEN
				// Success... Next station
				iPathID := iPathID + 1;
			ELSIF (iRes = 3) THEN
				// Error!
				// TODO!!!
				;
			END_IF
			
		ELSE
			iPathID := iPathID + 1;
		END_IF
		IF (iPathID >= MM_MAX_NUMBER_OF_PATH_ELEMENTS) THEN
			// All reset
			iPathID := 1;
			eTrackState := E_TrackState.ResetWait;
		END_IF

	E_TrackState.ResetWait:
		tonResetTime(IN := TRUE, PT := T#4S);
		IF (tonResetTime.Q) THEN
			tonResetTime(IN := FALSE);
			eTrackState := E_TrackState.ResetCheck;						
		END_IF
	
	E_TrackState.ResetCheck:
		IF (abControlledPaths[iPathID]) THEN
			// Is this path controlled by this cell
			IF (aReadPathData[iPathID].stPathData.bPathPresent AND
				( (aReadPathData[iPathID].stPathData.nState = E_MMPathState.eMMPathState_Operational) OR (aReadPathData[iPathID].stPathData.nState = E_MMPathState.eMMPathState_Initialization) )) THEN
				// This path is operational or reset completed
				bPathsReset := bPathsReset AND TRUE;
			ELSE
				// Not operational
				bPathsReset := FALSE;
			END_IF
		END_IF
		iPathID := iPathID + 1;
		IF (iPathID > MM_MAX_NUMBER_OF_PATH_ELEMENTS) THEN
			IF (bPathsReset) THEN
				// All paths OK... Continue
				iPathID := 1;
				eTrackState := E_TrackState.Idle;
			ELSIF (NOT bEnable) THEN
				// Stop
				eTrackState := E_TrackState.Undefined;			
			ELSE
				// All paths NOT OK!
				bPathsReset := TRUE;
				iPathID := 1;
			END_IF
		END_IF

	E_TrackState.Idle:
		IF (bEnable) THEN
			eTrackState := E_TrackState.Undefined;
		END_IF

	E_TrackState.Error:

END_CASE

tonSkipPathRead(IN := (eTrackState = E_TrackState.Started),
				PT := T#5S,
				Q => ,
				ET =>	);

// Shut down track from OPC-UA interface
IF (stAdditionalDataIn.bShutDown) THEN
	stAdditionalDataIn.bShutDown := FALSE;
	bEnable := FALSE;
END_IF
END_METHOD

METHOD PROTECTED M_StateMachineMethod : BOOL
VAR_INPUT
END_VAR
CASE eStateMethod OF
	E_TrackClientState.Disconnected:
		bConnectedMethod := FALSE;
		bBusyMethod := FALSE;
		fbConnectMethod.Execute := FALSE;
		fbDisconnectMethod.Execute := FALSE;
		fbGetNamespaceMethod.Execute := FALSE;
		fbGetHandleMethod.Execute := FALSE;
		fbCallMethod.Execute := FALSE;
		fbReleaseHandleMethod.Execute := FALSE;
		IF (bEnable) THEN
			bErrorMethod := FALSE;
			nErrorMethodID := 0;
			eStateMethod := E_TrackClientState.Connecting;
		END_IF
	
	E_TrackClientState.Connecting:
		IF (fbConnectMethod.Execute AND NOT fbConnectMethod.Busy) THEN
			fbConnectMethod.Execute := FALSE;
			IF (NOT fbConnectMethod.Error) THEN
				(* Connected *)
				nConnectHdlMethod := fbConnectMethod.ConnectionHdl;
				eStateMethod := E_TrackClientState.GetNamespaceIndex;
			ELSE
				(* Error during connection *)
				bErrorMethod := TRUE;
				nErrorMethodID := fbConnectMethod.ErrorID;
				eLastErrorMethodID := nErrorMethodID;
				nConnectHdlMethod := 0;
				eStateMethod := E_TrackClientState.Error;
			END_IF
		ELSE
			fbConnectMethod.Execute := TRUE;		
		END_IF
	
	E_TrackClientState.GetNamespaceIndex:
		IF (fbGetNamespaceMethod.Execute AND NOT fbGetNamespaceMethod.Busy) THEN
			fbGetNamespaceMethod.Execute := FALSE;
			IF (NOT fbGetNamespaceMethod.Error) THEN
				nNameSpaceIndexMethod := fbGetNamespaceMethod.NamespaceIndex;
				eStateMethod := E_TrackClientState.Connected;
			ELSE
				(* Error during get namepsace index *)
				nNameSpaceIndexMethod := 0;
				bErrorMethod := TRUE;
				nErrorMethodID := fbGetNamespaceMethod.ErrorID;
				eStateMethod := E_TrackClientState.Disconnecting;
			END_IF
		ELSE
			fbGetNamespaceMethod.Execute := TRUE;
		END_IF
	
	E_TrackClientState.Connected:
		bConnectedMethod := TRUE;
		bBusyMethod := FALSE;
		IF (NOT bEnable) THEN
			bConnectedMethod := FALSE;
			eStateMethod := E_TrackClientState.Disconnecting;
		ELSIF (bCallMethod) THEN
			bCallMethod := FALSE;
			bBusyMethod := TRUE;
			eStateMethod := E_TrackClientState.GetHandle;
		END_IF
		
	E_TrackClientState.GetHandle:
		IF (fbGetHandleMethod.Execute AND NOT fbGetHandleMethod.Busy) THEN
			fbGetHandleMethod.Execute := FALSE;
			IF (NOT fbGetHandleMethod.Error) THEN
				nHandleMethod := fbGetHandleMethod.MethodHdl;
				eStateMethod := E_TrackClientState.Execute;
			ELSE
				(* Error during get method handle *)
				nHandleMethod := 0;
				bErrorMethod := TRUE;
				nErrorMethodID := fbGetHandleMethod.ErrorID;
				eStateMethod := E_TrackClientState.Disconnecting;
			END_IF
		ELSE
			fbGetHandleMethod.Execute := TRUE;
		END_IF

	E_TrackClientState.Execute:
		IF (fbCallMethod.Execute AND NOT fbCallMethod.Busy) THEN
			fbCallMethod.Execute := FALSE;
			IF (NOT fbCallMethod.Error) THEN
				eStateMethod := E_TrackClientState.ReleaseHandle;
			ELSE
				(* Error during get namespace index *)
				bErrorMethod := TRUE;
				nErrorMethodID := fbCallMethod.ErrorID;
				eStateMethod := E_TrackClientState.ReleaseHandle;
			END_IF
		ELSE
			fbCallMethod.Execute := TRUE;
		END_IF
	
	E_TrackClientState.ReleaseHandle:
		IF (fbReleaseHandleMethod.Execute AND NOT fbReleaseHandleMethod.Busy) THEN
			fbReleaseHandleMethod.Execute := FALSE;
			IF (bErrorMethod) THEN
				eStateMethod := E_TrackClientState.Error;	
				nHandleMethod := 0;
			ELSIF (NOT fbReleaseHandleMethod.Error) THEN
				nHandleMethod := 0;
				eStateMethod := E_TrackClientState.Connected;
			ELSE
				(* Error during release handle *)
				bErrorMethod := TRUE;
				nErrorMethodID := fbReleaseHandleMethod.ErrorID;
				nHandleMethod := 0;
				eStateMethod := E_TrackClientState.Disconnecting;
			END_IF
		ELSE
			fbReleaseHandleMethod.Execute := TRUE;
		END_IF
	
	E_TrackClientState.Disconnecting:
		bConnectedMethod := FALSE;
		IF (fbDisconnectMethod.Execute AND NOT fbDisconnectMethod.Busy) THEN
			fbDisconnectMethod.Execute := FALSE;
			IF (bErrorMethod) THEN
				eStateMethod := E_TrackClientState.Error;	
				nConnectHdlMethod := 0;				
			ELSIF (NOT fbDisconnectMethod.Error) THEN
				(* Disconnected *)
				nConnectHdlMethod := 0;
				eStateMethod := E_TrackClientState.Disconnected;
			ELSE
				(* Error during disconnection *)
				bErrorMethod := TRUE;
				nErrorMethodID := fbDisconnectMethod.ErrorID;
				nConnectHdlMethod := 0;
				eStateMethod := E_TrackClientState.Error;
			END_IF
		ELSE
			fbDisconnectMethod.Execute := TRUE;
		END_IF
	
	E_TrackClientState.Error:
		eStateMethod := E_TrackClientState.Disconnected;
		
END_CASE
END_METHOD

METHOD PROTECTED M_StateMachineNode_ADS : INT
VAR_INPUT
END_VAR
CASE eStateNode OF
	E_TrackClientState.Disconnected:
		bConnectedNode := FALSE;
		fbReadADS( bEnable := FALSE ); 
		IF (bEnable) THEN
			bErrorNode := FALSE;
			nErrorNodeID := 0;
			eStateNode := E_TrackClientState.Connected;
		END_IF
	
	E_TrackClientState.Connecting:
		eStateNode := E_TrackClientState.GetNamespaceIndex;
	
	E_TrackClientState.GetNamespaceIndex:
		eStateNode := E_TrackClientState.Connected;
	
	E_TrackClientState.Connected:	
//		bConnectedNode := TRUE;
		IF (NOT bEnable) THEN
			bConnectedNode := FALSE;
			eStateNode := E_TrackClientState.Disconnecting;
		ELSIF (M_InitNodeData_ADS()) THEN
			eStateNode := E_TrackClientState.Execute;			
		END_IF
		
	E_TrackClientState.GetHandle:
		eStateNode := E_TrackClientState.Execute;
	
	E_TrackClientState.Execute:
		fbReadADS(	bEnable:= TRUE, 
							eType:= E_ADS_Comm_Type.ADS_RD_FAST, 
							rInterval:= rReadInterval, 
							pLocalVar:= pReadNodeData, // M_InitNodeData_ADS 
							nLocalSize:= UDINT_TO_UINT(cbDataTotal), // M_InitNodeData_ADS
							sNetID:= sTrackServerNetID, 
							nPort:= nTrackServerPortNo, 
							sVarName:= sTrackServerSymbol, // M_InitNodeData_ADS
							bWriteError=> , 
							bReadError=> , 
							bParameterError=> );
		IF (fbReadADS.bReadError OR fbReadADS.bParameterError) THEN
			eStateNode := E_TrackClientState.Error;			
		ELSIF (fbReadADS.M_SendRecvCompleted()) THEN
			bConnectedNode := TRUE;
			fbReadADS( bEnable := FALSE );
			IF (bReadDecPointVehicleBusy) THEN
				// Reading of decision point vehicle data has completed! 
				bReadDecPointVehicleBusy := FALSE;
			
			ELSIF (eReadType = E_OPC_NodeType.Stations) THEN
				// Reading stations
				IF (F_StringCompNoCase(aReadStationData[iReadIndex].stStationData.sCellID, sCellID)) THEN
					// The read station belongs to this cell
					FOR iStatIndex := 1 TO 5 BY 1 DO
						 IF (aStations[iStatIndex].bPresent) THEN
							// Station is present, check station ID against the read station ID
							IF (F_StringCompNoCase(aReadStationData[iReadIndex].stStationData.sStationID, aStations[iStatIndex].sStationID)) THEN
								// Found matching station ID. Store it...
								iThisStationIndex[iStatIndex] := iReadIndex;
							END_IF
						ELSE
							iThisStationIndex[iStatIndex] := 0;
						END_IF
					END_FOR
				END_IF
			
			ELSIF (bReadDecPointCell) THEN
				// Reading cell data completed
				bReadDecPointCell := FALSE;
				bReadDecPointCellDone := TRUE;
			
			END_IF
			
			eStateNode := E_TrackClientState.Connected;
			iLastReadTimeMS := iReadTimeMS;
			iReadTimeMS := 0;
		END_IF
	
	E_TrackClientState.ReleaseHandle:
		eStateNode := E_TrackClientState.Connected;
	
	E_TrackClientState.Disconnecting:
		bConnectedNode := FALSE;
		eStateNode := E_TrackClientState.Disconnected;
	
	E_TrackClientState.Error:
		tonErrorReset.IN := TRUE;
		IF (tonErrorReset.Q) THEN
			tonErrorReset.IN := FALSE;
			eStateNode := E_TrackClientState.Disconnected;
		END_IF
		
END_CASE

// Read timer
iReadTimeMS := iReadTimeMS + 10;
END_METHOD

METHOD PROTECTED M_ThisCellDataIndex : UINT
VAR_INPUT
END_VAR
VAR
	i		: UINT;
END_VAR
// Locate the status data for this cell!

(*
// Check if a value is already found
IF (iThisCellIndex > 0) THEN 
	// Check previous found value
	IF (F_StringCompNoCase(	s1 := sCellID, s2 := aReadCellData[iThisCellIndex].stCell.sCellID)) THEN
		// Previous found value is OK
		;
	ELSE
		// Previous found value is NOT OK, find correct value
		iThisCellIndex := 0;
	END_IF
END_IF

IF (iThisCellIndex = 0) THEN 
	// Find correct value
	FOR i := 1 TO MM_MAX_NUMBER_OF_STATION_ELEMENTS BY 1 DO
		IF (F_StringCompNoCase(sCellID, s2 := aReadCellData[i].stCell.sCellID)) THEN
			// Correct cell ID found
			iThisCellIndex := i;
			EXIT;
		END_IF
	END_FOR
END_IF
*)

M_ThisCellDataIndex := iThisCellIndex;
END_METHOD

METHOD PROTECTED M_UpdateStatus : BOOL
VAR_INPUT
END_VAR
VAR
	iBuffer				: UINT;
	iVehicleID			: UINT;
	iVehicleIndex		: UINT;
	bDataChanged		: BOOL;
END_VAR
// Update status values

// Check if LC allows to change status data
IF (stAdditionalDataIn.MESHandShakes.DataChangeStatusTransportStatus = stStatus.DataChange) THEN
	////////////////////////////////////////////////////////////////////////////////////////////////////////////////////////////////////
	// Vehicles
	////////////////////////////////////////////////////////////////////////////////////////////////////////////////////////////////////
	iVehicleIndex := 1;
	iVehicleID := 1;
	bDataChanged := FALSE;
	MEMSET(ADR(stStatus.Carrier), 0, SIZEOF(stStatus.Carrier));
	WHILE iVehicleID < MM_MAX_NUMBER_OF_VEHICLE_ELEMENTS DO
	
		IF ((aReadVehicleData[iVehicleID].stVehicle.nVehicleID > 0) AND
			(aReadVehicleData[iVehicleID].stVehicle.bDataValid) ) THEN
			// Vehicle has valid data
			IF ((aReadVehicleData[iVehicleID].stVehicle.sOwnerCell = sCellID) AND M_CheckVehicleOwned(aReadVehicleData[iVehicleID].stVehicle.nVehicleID)) THEN
				// Vehicle belongs to this cell
				stStatus.Carrier[iVehicleIndex].CarrierID := aReadVehicleData[iVehicleID].stVehicle.sCarrierID;
				stStatus.Carrier[iVehicleIndex].CarriersInPackage := aReadVehicleData[iVehicleID].stVehicle.nTicketSize; 
				stStatus.Carrier[iVehicleIndex].CarrierStatus := aReadVehicleData[iVehicleID].stVehicle.nState;
				stStatus.Carrier[iVehicleIndex].CurrentPath := aReadVehicleData[iVehicleID].stVehicle.nPathID;
				stStatus.Carrier[iVehicleIndex].CurrentPosition := aReadVehicleData[iVehicleID].stVehicle.fPosition;
				stStatus.Carrier[iVehicleIndex].CurrentStation := aReadVehicleData[iVehicleID].stVehicle.sCurrentStationID;
				stStatus.Carrier[iVehicleIndex].JobID := aReadVehicleData[iVehicleID].stVehicle.sJobID;
				IF (aReadVehicleData[iVehicleID].stVehicle.sLastScan <> '') THEN
					stStatus.Carrier[iVehicleIndex].LastScan := STRING_TO_DT(CONCAT('DT#', aReadVehicleData[iVehicleID].stVehicle.sLastScan));
				END_IF
				stStatus.Carrier[iVehicleIndex].Material := aReadVehicleData[iVehicleID].stVehicle.bMaterial;
				stStatus.Carrier[iVehicleIndex].MaterialID := aReadVehicleData[iVehicleID].stVehicle.sMaterialID;
				stStatus.Carrier[iVehicleIndex].Priority := aReadVehicleData[iVehicleID].stVehicle.nPriority;
				IF (aReadVehicleData[iVehicleID].stVehicle.sTargetStationID <> '') THEN
					stStatus.Carrier[iVehicleIndex].TargetReached := (aReadVehicleData[iVehicleID].stVehicle.sTargetStationID = aReadVehicleData[iVehicleID].stVehicle.sCurrentStationID);
				ELSE
					stStatus.Carrier[iVehicleIndex].TargetReached := FALSE;
				END_IF
				// Update Target Reached Counter
				IF ((aOldVehicleData[iVehicleID].sCurrentStationID = '') AND (aReadVehicleData[iVehicleID].stVehicle.sCurrentStationID <> '')) THEN
					IF (aReadVehicleData[iVehicleID].stVehicle.sTargetStationID = aReadVehicleData[iVehicleID].stVehicle.sCurrentStationID) THEN
						// First scan this vehicle is on position
						aOldVehicleTargetReachedCnt[iVehicleID] := aOldVehicleTargetReachedCnt[iVehicleID] + 1;
						IF (aOldVehicleTargetReachedCnt[iVehicleID] >= 100) THEN
							aOldVehicleTargetReachedCnt[iVehicleID] := 0;
						END_IF
					END_IF
				END_IF
				stStatus.Carrier[iVehicleIndex].TargetReachedCounter := (iThisCellIndex * 100) + aOldVehicleTargetReachedCnt[iVehicleID];
				stStatus.Carrier[iVehicleIndex].TargetStation := aReadVehicleData[iVehicleID].stVehicle.sTargetStationID;
				stStatus.Carrier[iVehicleIndex].Ticket := aReadVehicleData[iVehicleID].stVehicle.nTicket;
				stStatus.Carrier[iVehicleIndex].Tool := aReadVehicleData[iVehicleID].stVehicle.bTool;
				stStatus.Carrier[iVehicleIndex].ToolID := aReadVehicleData[iVehicleID].stVehicle.sToolID;
				stStatus.Carrier[iVehicleIndex].ValidData := aReadVehicleData[iVehicleID].stVehicle.bDataValid;
				stStatus.Carrier[iVehicleIndex].NOK := aReadVehicleData[iVehicleID].stVehicle.bNOK;
				
				iVehicleIndex := iVehicleIndex + 1;
				
				// Compare with old vehicle data
				bDataChanged := bDataChanged OR M_UpdateStatusCompare(iVehicleID);
			END_IF
		END_IF
	
		// Save as old vehicle data
		aOldVehicleData[iVehicleID] := aReadVehicleData[iVehicleID].stVehicle;
		
		// Next vehicle
		iVehicleID := iVehicleID + 1;
	END_WHILE
	stStatus.NumberOfCarriers := (iVehicleIndex - 1);
	// Check if number of carriers has changed and update data if it has
	IF (stStatus.NumberOfCarriers <> iOldVehicleCount) THEN
		bDataChanged := TRUE;
		iOldVehicleCount := stStatus.NumberOfCarriers;
	END_IF
	
	// Check if data has changed
	IF (bDataChanged OR bForceVehicleUpdateOPC) THEN
		bForceVehicleUpdateOPC := FALSE;
		stStatus.DataChange := stStatus.DataChange + 1;
	END_IF
	
	
	////////////////////////////////////////////////////////////////////////////////////////////////////////////////////////////////////
	// Stations
	////////////////////////////////////////////////////////////////////////////////////////////////////////////////////////////////////
	iStation := iStation + 1;
	IF (iStation > 5) THEN
		iStation := 1;
	END_IF
	// Station ID
	stStatus.StationBuffer[iStation].StationID := aStations[iStation].sStationID;
	IF (aStations[iStation].bPresent) THEN
		// Station 1 (input) values (placed at the first Pre-buffer index!)
		stStatus.StationBuffer[iStation].PreBuffer.BufferIndex[1].Present := aStations[iStation].stStationData1.bPresent;
		stStatus.StationBuffer[iStation].PreBuffer.BufferIndex[1].CarrierID := M_VehicleIDToCarrierID(aStations[iStation].stStationData1.nCurrentVehicleID);
		stStatus.StationBuffer[iStation].PreBuffer.BufferIndex[1].Ticket := aStations[iStation].stStationData1.nTicket;
		// Station 2 (output) values (placed at the first Post-buffer index!)
		stStatus.StationBuffer[iStation].PostBuffer.BufferIndex[1].Present := aStations[iStation].stStationData2.bPresent;
		stStatus.StationBuffer[iStation].PostBuffer.BufferIndex[1].CarrierID := M_VehicleIDToCarrierID(aStations[iStation].stStationData2.nCurrentVehicleID);
		stStatus.StationBuffer[iStation].PostBuffer.BufferIndex[1].Ticket := aStations[iStation].stStationData2.nTicket;
		// Buffers
		stStatus.StationBuffer[iStation].PreBuffer.Capacity := 0;
		stStatus.StationBuffer[iStation].PreBuffer.CapacityUsed := 0;
		stStatus.StationBuffer[iStation].PostBuffer.Capacity := 0;
		stStatus.StationBuffer[iStation].PostBuffer.CapacityUsed := 0;
		FOR iBuffer := 1 TO MM_MAX_BUFFER_INDEX BY 1 DO
			// Pre-buffer capacity
			IF (aStations[iStation].astPreBuffer[iBuffer].bPresent) THEN
				stStatus.StationBuffer[iStation].PreBuffer.Capacity := stStatus.StationBuffer[iStation].PreBuffer.Capacity + 1;
			END_IF
			// Pre-buffer used capacity
			IF (aStations[iStation].astPreBuffer[iBuffer].nCurrentVehicleID > 0) THEN
				stStatus.StationBuffer[iStation].PreBuffer.CapacityUsed := stStatus.StationBuffer[iStation].PreBuffer.CapacityUsed + 1;
			END_IF
			// Pre-buffer values
			stStatus.StationBuffer[iStation].PreBuffer.BufferIndex[iBuffer+1].Present := aStations[iStation].astPreBuffer[iBuffer].bPresent;
			stStatus.StationBuffer[iStation].PreBuffer.BufferIndex[iBuffer+1].CarrierID := M_VehicleIDToCarrierID(aStations[iStation].astPreBuffer[iBuffer].nCurrentVehicleID);
			stStatus.StationBuffer[iStation].PreBuffer.BufferIndex[iBuffer+1].Ticket := aStations[iStation].astPreBuffer[iBuffer].nTicket;
			// Post-buffer capacity
			IF (aStations[iStation].astPostBuffer[iBuffer].bPresent) THEN
				stStatus.StationBuffer[iStation].PostBuffer.Capacity := stStatus.StationBuffer[iStation].PostBuffer.Capacity + 1;
			END_IF
			// Post-buffer used capacity
			IF (aStations[iStation].astPostBuffer[iBuffer].nCurrentVehicleID > 0) THEN
				stStatus.StationBuffer[iStation].PostBuffer.CapacityUsed := stStatus.StationBuffer[iStation].PostBuffer.CapacityUsed + 1;
			END_IF
			// Post-buffer values
			stStatus.StationBuffer[iStation].PostBuffer.BufferIndex[iBuffer+1].Present := aStations[iStation].astPostBuffer[iBuffer].bPresent;
			stStatus.StationBuffer[iStation].PostBuffer.BufferIndex[iBuffer+1].CarrierID := M_VehicleIDToCarrierID(aStations[iStation].astPostBuffer[iBuffer].nCurrentVehicleID);
			stStatus.StationBuffer[iStation].PostBuffer.BufferIndex[iBuffer+1].Ticket := aStations[iStation].astPostBuffer[iBuffer].nTicket;
			
		END_FOR
	END_IF

END_IF
END_METHOD

/// Compares two vehicle data sets. Returns TRUE if different
METHOD PROTECTED M_UpdateStatusCompare : BOOL
VAR_INPUT
	iVehicleID		: UINT;
END_VAR

